# B&R Automation Studio project KeePakST401VersionX (part 2)

#### InverterFaultText.st - Implementation code
```iecst
(********************************************************************
 * COPYRIGHT --
 ********************************************************************
 * Program: ErrTxt
 * File: ErrTxt.st
 * Author: scoccimaroj
 * Created: November 09, 2010
 ********************************************************************
 * Implementation of function InverterFaultText
 ********************************************************************)

FUNCTION_BLOCK InverterFaultText

(*****************************************************************
		Initializing the Fault Tables
 ****************************************************************)

	IF ( isInitialized = FALSE) THEN
        (*ensure the fault table array creation is only run once upon start up*)
		isInitialized := TRUE;
        (*initialize internal fault comparison variable so that the first error is correctly written by the FUB *)
		PreviousFault :=  -1;
        (*initialize the output variable value*)
        LastFault := 0;
        (*this status will most likely not be seen by the FUB user but is written in case the table creation arrays are expanded enough for a visible delay to be seen*)
	    Status := INITIALIZING_ERROR_TEXT;

		(* Initialize the S44 Fault table first *)
		S44FaultTable[0].FaultNumber := 0;
		strcpy( ADR(S44FaultTable[0].FaultDescription), ADR('nOF - No Fault Present') );

		S44FaultTable[1].FaultNumber := 1;
		strcpy( ADR(S44FaultTable[1].FaultDescription), ADR('InF - Calibration Error') );

		S44FaultTable[2].FaultNumber := 3;
		strcpy( ADR(S44FaultTable[2].FaultDescription), ADR('CFF - Incorrect Configuration') );

		S44FaultTable[3].FaultNumber := 4;
		strcpy( ADR(S44FaultTable[3].FaultDescription), ADR('CFI - Invalid Configuration') );

		S44FaultTable[4].FaultNumber := 5;
		strcpy( ADR(S44FaultTable[4].FaultDescription), ADR('SLF1 - ModBus Communication Fault') );

		S44FaultTable[5].FaultNumber := 9;
		strcpy( ADR(S44FaultTable[5].FaultDescription), ADR('OCF - Over Current Fault') );

		S44FaultTable[6].FaultNumber := 10;
		strcpy( ADR(S44FaultTable[6].FaultDescription), ADR('CrF1 - Precharge Fault') );

		S44FaultTable[7].FaultNumber := 16;
		strcpy( ADR(S44FaultTable[7].FaultDescription), ADR('OHF - Drive Overheat') );

		S44FaultTable[8].FaultNumber := 17;
		strcpy( ADR(S44FaultTable[8].FaultDescription), ADR('OLF - Motor Overload') );

		S44FaultTable[9].FaultNumber := 18;
		strcpy( ADR(S44FaultTable[9].FaultDescription), ADR('ObF - Overbraking') );

		S44FaultTable[10].FaultNumber := 19;
		strcpy( ADR(S44FaultTable[10].FaultDescription), ADR('OSF - Mains Overvoltage') );

		S44FaultTable[11].FaultNumber := 20;
		strcpy( ADR(S44FaultTable[11].FaultDescription), ADR('OPF1 - 1 Output Phase Loss') );

		S44FaultTable[12].FaultNumber := 21;
		strcpy( ADR(S44FaultTable[12].FaultDescription), ADR('PHF - Input Phase Loss') );

		S44FaultTable[13].FaultNumber := 22;
		strcpy( ADR(S44FaultTable[13].FaultDescription), ADR('USF - Undervoltage') );

		S44FaultTable[14].FaultNumber := 23;
		strcpy( ADR(S44FaultTable[14].FaultDescription), ADR('SCF1 - Motor Short Circuit') );

		S44FaultTable[15].FaultNumber := 24;
		strcpy( ADR(S44FaultTable[15].FaultDescription), ADR('SOF - Overspeed') );

		S44FaultTable[16].FaultNumber := 25;
		strcpy( ADR(S44FaultTable[16].FaultDescription), ADR('tnF - Auto-tuning Fault') );

		S44FaultTable[17].FaultNumber := 26;
		strcpy( ADR(S44FaultTable[17].FaultDescription), ADR('InF1 - Rating Error') );

		S44FaultTable[18].FaultNumber := 27;
		strcpy( ADR(S44FaultTable[18].FaultDescription), ADR('InF2 - Power Calibration') );

		S44FaultTable[19].FaultNumber := 28;
		strcpy( ADR(S44FaultTable[19].FaultDescription), ADR('InF3 - Internal Serial Link') );

		S44FaultTable[20].FaultNumber := 29;
		strcpy( ADR(S44FaultTable[20].FaultDescription), ADR('InF4 - Internal Mfg area') );

		S44FaultTable[21].FaultNumber := 32;
		strcpy( ADR(S44FaultTable[21].FaultDescription), ADR('SCF3 - Ground Short Circuit') );

		S44FaultTable[22].FaultNumber := 33;
		strcpy( ADR(S44FaultTable[22].FaultDescription), ADR('OPF2 - 3 Output Phase Loss') );

		S44FaultTable[23].FaultNumber := 42;
		strcpy( ADR(S44FaultTable[23].FaultDescription), ADR('SLF2 - PowerSuite Communication') );

		S44FaultTable[24].FaultNumber := 45;
		strcpy( ADR(S44FaultTable[24].FaultDescription), ADR('SLF3 - HMI Communication Fault') );

		S44FaultTable[25].FaultNumber := 51;
		strcpy( ADR(S44FaultTable[25].FaultDescription), ADR('InF9 - Internal I measure') );

		S44FaultTable[26].FaultNumber := 53;
		strcpy( ADR(S44FaultTable[26].FaultDescription), ADR('InFb - Internal th. sensor') );

		S44FaultTable[27].FaultNumber := 54;
		strcpy( ADR(S44FaultTable[27].FaultDescription), ADR('tJF - IGBT Overheat') );

		S44FaultTable[28].FaultNumber := 55;
		strcpy( ADR(S44FaultTable[28].FaultDescription), ADR('SCF4 - IGBT Short Circuit') );

		S44FaultTable[29].FaultNumber := 56;
		strcpy( ADR(S44FaultTable[29].FaultDescription), ADR('SCF5 - Motor Short Circuit') );

		S44FaultTable[30].FaultNumber := 69;
		strcpy( ADR(S44FaultTable[30].FaultDescription), ADR('InFE - Internal CPU Fault') );

		S44FaultTable[31].FaultNumber := 77;
		strcpy( ADR(S44FaultTable[31].FaultDescription), ADR('CFI2') );

		S44FaultTable[32].FaultNumber := 100;
		strcpy( ADR(S44FaultTable[32].FaultDescription), ADR('ULF - Underload Fault') );

		S44FaultTable[33].FaultNumber := 101;
		strcpy( ADR(S44FaultTable[33].FaultDescription), ADR('OLC - Overload Fault') );

		S44FaultTable[34].FaultNumber := 106;
		strcpy( ADR(S44FaultTable[34].FaultDescription), ADR('LFF1') );

		S44FaultTable[35].FaultNumber := 253;
		strcpy( ADR(S44FaultTable[35].FaultDescription), ADR('XXXX') );

		(* Initialize the X64 Table *)
		X64FaultTable[0].FaultNumber := 0;
		strcpy( ADR(X64FaultTable[0].FaultDescription), ADR('nOF - No Fault Code') );

		X64FaultTable[1].FaultNumber := 3;
		strcpy( ADR(X64FaultTable[1].FaultDescription), ADR('CFF - Incorrect Configuration') );

		X64FaultTable[2].FaultNumber := 4;
		strcpy( ADR(X64FaultTable[2].FaultDescription), ADR('CFI - Invalid Configuration') );

		X64FaultTable[3].FaultNumber := 5;
		strcpy( ADR(X64FaultTable[3].FaultDescription), ADR('SLF - Communication Fault') );

		X64FaultTable[4].FaultNumber := 6;
		strcpy( ADR(X64FaultTable[4].FaultDescription), ADR('ILF - Internal Communication Interuption') );

		X64FaultTable[5].FaultNumber := 7;
		strcpy( ADR(X64FaultTable[5].FaultDescription), ADR('CnF - Communication Option Card') );

		X64FaultTable[6].FaultNumber := 8;
		strcpy( ADR(X64FaultTable[6].FaultDescription), ADR('EPF - External Fault') );

		X64FaultTable[7].FaultNumber := 9;
		strcpy( ADR(X64FaultTable[7].FaultDescription), ADR('OCF - Overcurrent') );

		X64FaultTable[8].FaultNumber := 10;
		strcpy( ADR(X64FaultTable[8].FaultDescription), ADR('CrF - Capacitor pre-charge') );

		X64FaultTable[9].FaultNumber := 13;
		strcpy( ADR(X64FaultTable[9].FaultDescription), ADR('LFF - 4 - 20 mA loss') );

		X64FaultTable[10].FaultNumber := 16;
		strcpy( ADR(X64FaultTable[10].FaultDescription), ADR('OHF - Drive Overheating') );

		X64FaultTable[11].FaultNumber := 17;
		strcpy( ADR(X64FaultTable[11].FaultDescription), ADR('OLF - Motor Overload') );

		X64FaultTable[12].FaultNumber := 18;
		strcpy( ADR(X64FaultTable[12].FaultDescription), ADR('ObF - DC Bus Overvoltage') );

		X64FaultTable[13].FaultNumber := 19;
		strcpy( ADR(X64FaultTable[13].FaultDescription), ADR('OSF - Line Supply Overvoltage') );

		X64FaultTable[14].FaultNumber := 20;
		strcpy( ADR(X64FaultTable[14].FaultDescription), ADR('OPF - Motor Phase Lose') );

		X64FaultTable[15].FaultNumber := 21;
		strcpy( ADR(X64FaultTable[15].FaultDescription), ADR('PHF - Line Phase Loss') );

		X64FaultTable[16].FaultNumber := 22;
		strcpy( ADR(X64FaultTable[16].FaultDescription), ADR('USF - Line Supply Undervoltage') );

		X64FaultTable[17].FaultNumber := 23;
		strcpy( ADR(X64FaultTable[17].FaultDescription), ADR('OCF - Motor Short Circuit (phase to phase)') );

		X64FaultTable[18].FaultNumber := 24;
		strcpy( ADR(X64FaultTable[18].FaultDescription), ADR('SOF - Motor Overspeed') );

		X64FaultTable[19].FaultNumber := 25;
		strcpy( ADR(X64FaultTable[19].FaultDescription), ADR('tnF - Auto-tuning was unsuccessful') );

		X64FaultTable[20].FaultNumber := 26;
		strcpy( ADR(X64FaultTable[20].FaultDescription), ADR('IF1 - Unknow rating') );

		X64FaultTable[21].FaultNumber := 27;
		strcpy( ADR(X64FaultTable[21].FaultDescription), ADR('IF2 - MMI card') );

		X64FaultTable[22].FaultNumber := 28;
		strcpy( ADR(X64FaultTable[22].FaultDescription), ADR('IF3 - MMI communication') );

		X64FaultTable[23].FaultNumber := 29;
		strcpy( ADR(X64FaultTable[23].FaultDescription), ADR('IF4 - Industrial EEPROM memory') );

		X64FaultTable[24].FaultNumber := 30;
		strcpy( ADR(X64FaultTable[24].FaultDescription), ADR('EEF - EEPROM memory') );

		X64FaultTable[25].FaultNumber := 31;
		strcpy( ADR(X64FaultTable[25].FaultDescription), ADR('OCF - Impeding Short Circuit') );

		X64FaultTable[26].FaultNumber := 32;
		strcpy( ADR(X64FaultTable[26].FaultDescription), ADR('SCF - Motor Short Circuit (to ground)') );

		X64FaultTable[27].FaultNumber := 33;
		strcpy( ADR(X64FaultTable[27].FaultDescription), ADR('OPF - Motor Phase Loss - 3 phases') );

		X64FaultTable[28].FaultNumber := 34;
		strcpy( ADR(X64FaultTable[28].FaultDescription), ADR('COF - Communication Interuption') );

		X64FaultTable[29].FaultNumber := 35;
		strcpy( ADR(X64FaultTable[29].FaultDescription), ADR('bLF - Brake Control') );

		X64FaultTable[30].FaultNumber := 36;
		strcpy( ADR(X64FaultTable[30].FaultDescription), ADR('OCF - Power Module on 15 kW drive') );

		X64FaultTable[31].FaultNumber := 55;
		strcpy( ADR(X64FaultTable[31].FaultDescription), ADR('SCF - Power Module or Motor Short Circuit') );

		(* Initialize the P84 Table *)
		P84FaultTable[0].FaultNumber := 0;
		strcpy( ADR(P84FaultTable[0].FaultDescription), ADR('nOF - No Fault') );

		P84FaultTable[1].FaultNumber := 1;
		strcpy( ADR(P84FaultTable[1].FaultDescription), ADR('InF - Calibration Error') );

		P84FaultTable[2].FaultNumber := 2;
		strcpy( ADR(P84FaultTable[2].FaultDescription), ADR('EEF1 - Control EEPROM') );

		P84FaultTable[3].FaultNumber := 3;
		strcpy( ADR(P84FaultTable[3].FaultDescription), ADR('CFF - Incorrect Configuration') );

		P84FaultTable[4].FaultNumber := 4;
		strcpy( ADR(P84FaultTable[4].FaultDescription), ADR('CFI - Invalid Configuration') );

		P84FaultTable[5].FaultNumber := 5;
		strcpy( ADR(P84FaultTable[5].FaultDescription), ADR('SLF1 - Communication Error') );

		P84FaultTable[6].FaultNumber := 6;
		strcpy( ADR(P84FaultTable[6].FaultDescription), ADR('ILF - Internal Communication Link') );

		P84FaultTable[7].FaultNumber := 7;
		strcpy( ADR(P84FaultTable[7].FaultDescription), ADR('CnF - Communication Network') );

		P84FaultTable[8].FaultNumber := 8;
		strcpy( ADR(P84FaultTable[8].FaultDescription), ADR('EPF1 - External Fault') );

		P84FaultTable[9].FaultNumber := 9;
		strcpy( ADR(P84FaultTable[9].FaultDescription), ADR('OCF - Overcurrent') );

		P84FaultTable[10].FaultNumber := 10;
		strcpy( ADR(P84FaultTable[10].FaultDescription), ADR('CrF - Precharge') );

		P84FaultTable[11].FaultNumber := 11;
		strcpy( ADR(P84FaultTable[11].FaultDescription), ADR('SPF - Speed Feedback loss') );

		P84FaultTable[12].FaultNumber := 12;
		strcpy( ADR(P84FaultTable[12].FaultDescription), ADR('AnF - Load Slipping') );

		P84FaultTable[13].FaultNumber := 13;
		strcpy( ADR(P84FaultTable[13].FaultDescription), ADR('LFF2 - AI2 4-20 mA Loss') );

		P84FaultTable[14].FaultNumber := 14;
		strcpy( ADR(P84FaultTable[14].FaultDescription), ADR('PtF1 - PTC1 Probe') );

		P84FaultTable[15].FaultNumber := 15;
		strcpy( ADR(P84FaultTable[15].FaultDescription), ADR('OtF1 - PTC1 Overheat') );

		P84FaultTable[16].FaultNumber := 16;
		strcpy( ADR(P84FaultTable[16].FaultDescription), ADR('OHF - Drive Overheat') );

		P84FaultTable[17].FaultNumber := 17;
		strcpy( ADR(P84FaultTable[17].FaultDescription), ADR('OLF - Motor Overload') );

		P84FaultTable[18].FaultNumber := 18;
		strcpy( ADR(P84FaultTable[18].FaultDescription), ADR('ObF - Overbraking') );

		P84FaultTable[19].FaultNumber := 19;
		strcpy( ADR(P84FaultTable[19].FaultDescription), ADR('OSF - Mains Overvoltage') );

		P84FaultTable[20].FaultNumber := 20;
		strcpy( ADR(P84FaultTable[20].FaultDescription), ADR('OPF1 - 1 Output Phase Loss') );

		P84FaultTable[21].FaultNumber := 21;
		strcpy( ADR(P84FaultTable[21].FaultDescription), ADR('PHF - Input Phase Loss') );

		P84FaultTable[22].FaultNumber := 22;
		strcpy( ADR(P84FaultTable[22].FaultDescription), ADR('USF - Undervoltage') );

		P84FaultTable[23].FaultNumber := 23;
		strcpy( ADR(P84FaultTable[23].FaultDescription), ADR('SCF1 - Motor Short Circuit') );

		P84FaultTable[24].FaultNumber := 24;
		strcpy( ADR(P84FaultTable[24].FaultDescription), ADR('SOF - Overspeed') );

		P84FaultTable[25].FaultNumber := 25;
		strcpy( ADR(P84FaultTable[25].FaultDescription), ADR('tnF - Auto-tuning Unsuccessful') );

		P84FaultTable[26].FaultNumber := 26;
		strcpy( ADR(P84FaultTable[26].FaultDescription), ADR('InF1 - Rating Error') );

		P84FaultTable[27].FaultNumber := 27;
		strcpy( ADR(P84FaultTable[27].FaultDescription), ADR('InF2 - Power Calibration') );

		P84FaultTable[28].FaultNumber := 28;
		strcpy( ADR(P84FaultTable[28].FaultDescription), ADR('InF3 - Internal Serial Link') );

		P84FaultTable[29].FaultNumber := 29;
		strcpy( ADR(P84FaultTable[29].FaultDescription), ADR('InF4 - Internal Mfg Area') );

		P84FaultTable[30].FaultNumber := 30;
		strcpy( ADR(P84FaultTable[30].FaultDescription), ADR('EEF2 - Power EEPROM') );

		P84FaultTable[31].FaultNumber := 31;
		strcpy( ADR(P84FaultTable[31].FaultDescription), ADR('SCF2 - Impedant Short Circuit') );

		P84FaultTable[32].FaultNumber := 32;
		strcpy( ADR(P84FaultTable[32].FaultDescription), ADR('SCF3 - Ground Short Circuit') );

		P84FaultTable[33].FaultNumber := 33;
		strcpy( ADR(P84FaultTable[33].FaultDescription), ADR('OPF2 - 3 Phase Output Loss') );

		P84FaultTable[34].FaultNumber := 34;
		strcpy( ADR(P84FaultTable[34].FaultDescription), ADR('COF - Powerlink Communication') );

		P84FaultTable[35].FaultNumber := 35;
		strcpy( ADR(P84FaultTable[35].FaultDescription), ADR('bLF - Brake Control') );

		P84FaultTable[36].FaultNumber := 37;
		strcpy( ADR(P84FaultTable[36].FaultDescription), ADR('InF7 - Internal Hard Init') );

		P84FaultTable[37].FaultNumber := 38;
		strcpy( ADR(P84FaultTable[37].FaultDescription), ADR('EPF2 - External Fault Com.') );

		P84FaultTable[38].FaultNumber := 39;
		strcpy( ADR(P84FaultTable[38].FaultDescription), ADR('APF - Application Fault') );

		P84FaultTable[39].FaultNumber := 40;
		strcpy( ADR(P84FaultTable[39].FaultDescription), ADR('InF8 - Internal Ctrl Supply') );

		P84FaultTable[40].FaultNumber := 41;
		strcpy( ADR(P84FaultTable[40].FaultDescription), ADR('brF - Brake Feedback') );

		P84FaultTable[41].FaultNumber := 42;
		strcpy( ADR(P84FaultTable[41].FaultDescription), ADR('SLF2 - PowerSuite Communication.') );

		P84FaultTable[42].FaultNumber := 43;
		strcpy( ADR(P84FaultTable[42].FaultDescription), ADR('ECF - Encoder Coupling') );

		P84FaultTable[43].FaultNumber := 44;
		strcpy( ADR(P84FaultTable[43].FaultDescription), ADR('SSF - Torque Current Limit') );

		P84FaultTable[44].FaultNumber :=45 ;
		strcpy( ADR(P84FaultTable[44].FaultDescription), ADR('SLF3 - HMI com.') );

		P84FaultTable[45].FaultNumber := 46;
		strcpy( ADR(P84FaultTable[45].FaultDescription), ADR('PrF - Power Removal') );

		P84FaultTable[46].FaultNumber := 47;
		strcpy( ADR(P84FaultTable[46].FaultDescription), ADR('PtF2 - PTC2 Probe') );

		P84FaultTable[47].FaultNumber := 48;
		strcpy( ADR(P84FaultTable[47].FaultDescription), ADR('OtF2 - PTC2 Overheat') );

		P84FaultTable[48].FaultNumber := 49;
		strcpy( ADR(P84FaultTable[48].FaultDescription), ADR('PtFL - LI6=PTC Probe') );

		P84FaultTable[49].FaultNumber := 50;
		strcpy( ADR(P84FaultTable[49].FaultDescription), ADR('OtFL - PTC Fault') );

		P84FaultTable[50].FaultNumber := 51;
		strcpy( ADR(P84FaultTable[50].FaultDescription), ADR('InF9 - Internal I measure') );

		P84FaultTable[51].FaultNumber := 52;
		strcpy( ADR(P84FaultTable[51].FaultDescription), ADR('InFA - Internal Mains Circuit') );

		P84FaultTable[52].FaultNumber := 53;
		strcpy( ADR(P84FaultTable[52].FaultDescription), ADR('InFb - Internal th. Sensor') );

		P84FaultTable[53].FaultNumber := 54;
		strcpy( ADR(P84FaultTable[53].FaultDescription), ADR('tJF - IGBT Overheat') );

		P84FaultTable[54].FaultNumber := 55;
		strcpy( ADR(P84FaultTable[54].FaultDescription), ADR('SCF4 - IGBT Short Circuit') );

		P84FaultTable[55].FaultNumber := 56;
		strcpy( ADR(P84FaultTable[55].FaultDescription), ADR('SCF5 - Motor Short Circuit') );

		P84FaultTable[56].FaultNumber :=57 ;
		strcpy( ADR(P84FaultTable[56].FaultDescription), ADR('SrF - Torque Time-out') );

		P84FaultTable[57].FaultNumber := 58;
		strcpy( ADR(P84FaultTable[57].FaultDescription), ADR('FCF1 - Output Contact Stuck') );

		P84FaultTable[58].FaultNumber := 59;
		strcpy( ADR(P84FaultTable[58].FaultDescription), ADR('FCF2 - Output Contact Open') );

		P84FaultTable[59].FaultNumber := 60;
		strcpy( ADR(P84FaultTable[59].FaultDescription), ADR('InFC - Int. T Measurement') );

		P84FaultTable[60].FaultNumber := 61;
		strcpy( ADR(P84FaultTable[60].FaultDescription), ADR('AI2F - AI2 Input') );

		P84FaultTable[61].FaultNumber := 62;
		strcpy( ADR(P84FaultTable[61].FaultDescription), ADR('EnF - Encoder') );

		P84FaultTable[62].FaultNumber := 63;
		strcpy( ADR(P84FaultTable[62].FaultDescription), ADR('CrF2 - Thyr. Soft Charge') );

		P84FaultTable[63].FaultNumber := 64;
		strcpy( ADR(P84FaultTable[63].FaultDescription), ADR('LCF - Input Contactor') );

		P84FaultTable[64].FaultNumber := 65;
		strcpy( ADR(P84FaultTable[64].FaultDescription), ADR('bUF - DB Unit Short Circuit') );

		P84FaultTable[65].FaultNumber := 66;
		strcpy( ADR(P84FaultTable[65].FaultDescription), ADR('dCF - Iff. I Fault') );

		P84FaultTable[66].FaultNumber := 67;
		strcpy( ADR(P84FaultTable[66].FaultDescription), ADR('HdF - IGBT  Desaturation') );

		P84FaultTable[67].FaultNumber := 68;
		strcpy( ADR(P84FaultTable[67].FaultDescription), ADR('InF6 - Internal Option') );

		P84FaultTable[68].FaultNumber := 69;
		strcpy( ADR(P84FaultTable[68].FaultDescription), ADR('InFE - Internal CPU') );

		P84FaultTable[69].FaultNumber := 70;
		strcpy( ADR(P84FaultTable[69].FaultDescription), ADR('bOF - BR Overload') );

		P84FaultTable[70].FaultNumber := 71;
		strcpy( ADR(P84FaultTable[70].FaultDescription), ADR('LFF3 - AI3 4-20 mA Loss') );

		P84FaultTable[71].FaultNumber := 72;
		strcpy( ADR(P84FaultTable[71].FaultDescription), ADR('LEF4 - AI4 4-20 mA Loss') );

		P84FaultTable[72].FaultNumber := 73;
		strcpy( ADR(P84FaultTable[72].FaultDescription), ADR('HCF - Cards Pairing') );

		P84FaultTable[73].FaultNumber := 76;
		strcpy( ADR(P84FaultTable[73].FaultDescription), ADR('dLF - Load Fault') );

		P84FaultTable[74].FaultNumber := 99;
		strcpy( ADR(P84FaultTable[74].FaultDescription), ADR('CSF - Ch. SW. Fault') );

		(* Initialize the P74 Table *)
		P74FaultTable[0].FaultNumber := 0;
		strcpy( ADR(P74FaultTable[0].FaultDescription), ADR('nOF - No Fault') );

		P74FaultTable[1].FaultNumber := 1;
		strcpy( ADR(P74FaultTable[1].FaultDescription), ADR('InF - Calibration Error') );

		P74FaultTable[2].FaultNumber := 2;
		strcpy( ADR(P74FaultTable[2].FaultDescription), ADR('EEF1 - Control EEPROM') );

		P74FaultTable[3].FaultNumber := 3;
		strcpy( ADR(P74FaultTable[3].FaultDescription), ADR('CFF - Incorrect Configuration') );

		P74FaultTable[4].FaultNumber := 4;
		strcpy( ADR(P74FaultTable[4].FaultDescription), ADR('CFI - Invalid Configuration') );

		P74FaultTable[5].FaultNumber := 5;
		strcpy( ADR(P74FaultTable[5].FaultDescription), ADR('SLF1 - Communication Error') );

		P74FaultTable[6].FaultNumber := 6;
		strcpy( ADR(P74FaultTable[6].FaultDescription), ADR('ILF - Internal Communication Link') );

		P74FaultTable[7].FaultNumber := 7;
		strcpy( ADR(P74FaultTable[7].FaultDescription), ADR('CnF - Communication Network') );

		P74FaultTable[8].FaultNumber := 8;
		strcpy( ADR(P74FaultTable[8].FaultDescription), ADR('EPF1 - External Fault') );

		P74FaultTable[9].FaultNumber := 9;
		strcpy( ADR(P74FaultTable[9].FaultDescription), ADR('OCF - Overcurrent') );

		P74FaultTable[10].FaultNumber := 10;
		strcpy( ADR(P74FaultTable[10].FaultDescription), ADR('CrF - Precharge') );

		P74FaultTable[11].FaultNumber := 11;
		strcpy( ADR(P74FaultTable[11].FaultDescription), ADR('SPF - Speed Feedback loss') );

		P74FaultTable[12].FaultNumber := 16;
		strcpy( ADR(P74FaultTable[12].FaultDescription), ADR('OHF - Drive Overheat') );

		P74FaultTable[13].FaultNumber := 17;
		strcpy( ADR(P74FaultTable[13].FaultDescription), ADR('OLF - Motor Overload') );

		P74FaultTable[14].FaultNumber := 18;
		strcpy( ADR(P74FaultTable[14].FaultDescription), ADR('ObF - Overbraking') );

		P74FaultTable[15].FaultNumber := 19;
		strcpy( ADR(P74FaultTable[15].FaultDescription), ADR('OSF - Mains Overvoltage') );

		P74FaultTable[16].FaultNumber := 20;
		strcpy( ADR(P74FaultTable[16].FaultDescription), ADR('OPF1 - 1 Output Phase Loss') );

		P74FaultTable[17].FaultNumber := 21;
		strcpy( ADR(P74FaultTable[17].FaultDescription), ADR('PHF - Input Phase Loss') );

		P74FaultTable[18].FaultNumber := 22;
		strcpy( ADR(P74FaultTable[18].FaultDescription), ADR('USF - Undervoltage') );

		P74FaultTable[19].FaultNumber := 23;
		strcpy( ADR(P74FaultTable[19].FaultDescription), ADR('SCF1 - Motor Short Circuit') );

		P74FaultTable[20].FaultNumber := 24;
		strcpy( ADR(P74FaultTable[20].FaultDescription), ADR('SOF - Overspeed') );

		P74FaultTable[21].FaultNumber := 25;
		strcpy( ADR(P74FaultTable[21].FaultDescription), ADR('tnF - Auto-tuning Unsuccessful') );

		P74FaultTable[22].FaultNumber := 26;
		strcpy( ADR(P74FaultTable[22].FaultDescription), ADR('InF1 - Rating Error') );

		P74FaultTable[23].FaultNumber := 27;
		strcpy( ADR(P74FaultTable[23].FaultDescription), ADR('InF2 - Power Calibration') );

		P74FaultTable[24].FaultNumber := 28;
		strcpy( ADR(P74FaultTable[24].FaultDescription), ADR('InF3 - Internal Serial Link') );

		P74FaultTable[25].FaultNumber := 29;
		strcpy( ADR(P74FaultTable[25].FaultDescription), ADR('InF4 - Internal Mfg Area') );

		P74FaultTable[26].FaultNumber := 30;
		strcpy( ADR(P74FaultTable[26].FaultDescription), ADR('EEF2 - Power EEPROM') );

		P74FaultTable[27].FaultNumber := 31;
		strcpy( ADR(P74FaultTable[27].FaultDescription), ADR('SCF2 - Impedant Short Circuit') );

		P74FaultTable[28].FaultNumber := 32;
		strcpy( ADR(P74FaultTable[28].FaultDescription), ADR('SCF3 - Ground Short Circuit') );

		P74FaultTable[29].FaultNumber := 33;
		strcpy( ADR(P74FaultTable[29].FaultDescription), ADR('OPF2 - 3 Phase Output Loss') );

		P74FaultTable[30].FaultNumber := 34;
		strcpy( ADR(P74FaultTable[30].FaultDescription), ADR('COF - Powerlink Communication') );

		P74FaultTable[31].FaultNumber := 35;
		strcpy( ADR(P74FaultTable[31].FaultDescription), ADR('bLF - Brake Control') );

		P74FaultTable[32].FaultNumber := 38;
		strcpy( ADR(P74FaultTable[32].FaultDescription), ADR('EPF2 - External Fault Com.') );

		P74FaultTable[33].FaultNumber := 41;
		strcpy( ADR(P74FaultTable[33].FaultDescription), ADR('brF - Brake Feedback') );

		P74FaultTable[34].FaultNumber := 42;
		strcpy( ADR(P74FaultTable[34].FaultDescription), ADR('SLF2 - PowerSuite Communication.') );

		P74FaultTable[35].FaultNumber := 43;
		strcpy( ADR(P74FaultTable[35].FaultDescription), ADR('ECF - Encoder Coupling') );

		P74FaultTable[36].FaultNumber := 44;
		strcpy( ADR(P74FaultTable[36].FaultDescription), ADR('SSF - Torque Current Limit') );

		P74FaultTable[37].FaultNumber := 45 ;
		strcpy( ADR(P74FaultTable[37].FaultDescription), ADR('SLF3 - HMI com.') );

		P74FaultTable[38].FaultNumber := 46;
		strcpy( ADR(P74FaultTable[38].FaultDescription), ADR('PrF - Power Removal') );

		P74FaultTable[39].FaultNumber := 49;
		strcpy( ADR(P74FaultTable[39].FaultDescription), ADR('PtFL - LI6=PTC Probe') );

		P74FaultTable[40].FaultNumber := 50;
		strcpy( ADR(P74FaultTable[40].FaultDescription), ADR('OtFL - PTC Fault') );

		P74FaultTable[41].FaultNumber := 51;
		strcpy( ADR(P74FaultTable[41].FaultDescription), ADR('InF9 - Internal I measure') );

		P74FaultTable[42].FaultNumber := 52;
		strcpy( ADR(P74FaultTable[42].FaultDescription), ADR('InFA - Internal Mains Circuit') );

		P74FaultTable[43].FaultNumber := 53;
		strcpy( ADR(P74FaultTable[43].FaultDescription), ADR('InFb - Internal th. Sensor') );

		P74FaultTable[44].FaultNumber := 54;
		strcpy( ADR(P74FaultTable[44].FaultDescription), ADR('tJF - IGBT Overheat') );

		P74FaultTable[45].FaultNumber := 55;
		strcpy( ADR(P74FaultTable[45].FaultDescription), ADR('SCF4 - IGBT Short Circuit') );

		P74FaultTable[46].FaultNumber := 56;
		strcpy( ADR(P74FaultTable[46].FaultDescription), ADR('SCF5 - Motor Short Circuit') );

		P74FaultTable[47].FaultNumber := 57 ;
		strcpy( ADR(P74FaultTable[47].FaultDescription), ADR('SrF - Torque Time-out') );

		P74FaultTable[48].FaultNumber := 58;
		strcpy( ADR(P74FaultTable[48].FaultDescription), ADR('FCF1 - Output Contact Stuck') );

		P74FaultTable[49].FaultNumber := 59;
		strcpy( ADR(P74FaultTable[49].FaultDescription), ADR('FCF2 - Output Contact Open') );

		P74FaultTable[50].FaultNumber := 61;
		strcpy( ADR(P74FaultTable[50].FaultDescription), ADR('AI2F - AI2 Input') );

		P74FaultTable[51].FaultNumber := 64;
		strcpy( ADR(P74FaultTable[51].FaultDescription), ADR('LCF - Input Contactor') );

		P74FaultTable[52].FaultNumber := 66;
		strcpy( ADR(P74FaultTable[52].FaultDescription), ADR('dCF - Iff. I Fault') );

		P74FaultTable[53].FaultNumber := 67;
		strcpy( ADR(P74FaultTable[53].FaultDescription), ADR('HdF - IGBT  Desaturation') );

		P74FaultTable[54].FaultNumber := 68;
		strcpy( ADR(P74FaultTable[54].FaultDescription), ADR('InF6 - Internal Option') );

		P74FaultTable[55].FaultNumber := 69;
		strcpy( ADR(P74FaultTable[55].FaultDescription), ADR('InFE - Internal CPU') );

		P74FaultTable[56].FaultNumber := 71;
		strcpy( ADR(P74FaultTable[56].FaultDescription), ADR('LFF3 - AI3 4-20 mA Loss') );

		P74FaultTable[57].FaultNumber := 73;
		strcpy( ADR(P74FaultTable[57].FaultDescription), ADR('HCF - Cards Pairing') );

		P74FaultTable[58].FaultNumber := 76;
		strcpy( ADR(P74FaultTable[58].FaultDescription), ADR('dLF - Load Fault') );

		P74FaultTable[59].FaultNumber := 77;
		strcpy( ADR(P74FaultTable[59].FaultDescription), ADR('CFI2 - Bad Configuration') );

		P74FaultTable[60].FaultNumber := 99;
		strcpy( ADR(P74FaultTable[60].FaultDescription), ADR('CSF - Ch. SW. Fault') );

		P74FaultTable[61].FaultNumber := 100;
		strcpy( ADR(P74FaultTable[61].FaultDescription), ADR('ULF - Pr. Underload Fault') );

		P74FaultTable[62].FaultNumber := 101;
		strcpy( ADR(P74FaultTable[62].FaultDescription), ADR('OLC - Proc. Overload Fault') );

		P74FaultTable[63].FaultNumber := 105;
		strcpy( ADR(P74FaultTable[63].FaultDescription), ADR('ASF - Angle Error') );

		P74FaultTable[64].FaultNumber := 107;
		strcpy( ADR(P74FaultTable[64].FaultDescription), ADR('SAFF - Safety Fault') );

		P74FaultTable[65].FaultNumber := 108;
		strcpy( ADR(P74FaultTable[65].FaultDescription), ADR('FbE - FB Fault') );

		P74FaultTable[66].FaultNumber := 109;
		strcpy( ADR(P74FaultTable[66].FaultDescription), ADR('FbES - FB Stop Fault') );
	ELSE
        (*this status will only be seen if the initialization of the fualt text arrays fails*)
        Status := INACTIVE;
	END_IF

	(* End of initializing the tables *)

	(*****************************************************
	Getting the Fault Text
	*****************************************************)
    IF isInitialized = TRUE THEN
        (* Do the search for a S44 drive *)
        IF (DriveType = EACPInverter_S44) THEN

            (*Cyclically write the internal previous fault number into the output variable LastFault*)
            LastFault := PreviousFault;

            IF Execute = TRUE THEN
                Status := BUSY;
                (* Only do a look up if a new fault number occured *)
                IF ( PreviousFault <> FaultNumber ) THEN
                    PreviousFault := FaultNumber;

                    (* Clear out the text in the fault string *)
                    strcpy(FaultText, ADR('') );

                    FOR i:= 0 TO 35 BY 1 DO
                        IF (FaultNumber = S44FaultTable[i].FaultNumber) THEN
                            strcpy(FaultText, ADR(S44FaultTable[i].FaultDescription) );
                            EXIT;
                        END_IF;
                    END_FOR;
                END_IF;
            ELSE
                Status := IDLE;
            END_IF;
            (* Do the search for a X64 drive *)
        ELSIF (DriveType = EACPInverter_X64) THEN

            (*Cyclically write the internal previous fault number into the output variable LastFault*)
            LastFault := PreviousFault;

            IF Execute = TRUE THEN
                Status := BUSY;
                (* Only do a look up if a new fault number occured *)
                IF ( PreviousFault <> FaultNumber ) THEN
                    PreviousFault := FaultNumber;

                    (* Clear out the text in the fault string *)
                    strcpy(FaultText, ADR('') );

                    FOR i:= 0 TO 31 BY 1 DO
                        IF (FaultNumber = X64FaultTable[i].FaultNumber) THEN
                            strcpy(FaultText, ADR(X64FaultTable[i].FaultDescription) );
                            EXIT;
                        END_IF;
                    END_FOR;
                END_IF;
            ELSE
                Status := IDLE;
            END_IF;

            (* Do the search for a P84 drive *)
        ELSIF (DriveType = EACPInverter_P84) THEN

            (*Cyclically write the internal previous fault number into the output variable LastFault*)
            LastFault := PreviousFault;

            IF Execute = TRUE THEN
                Status := BUSY;
                (* Only do a look up if a new fault number occured *)
                IF ( PreviousFault <> FaultNumber ) THEN
                    PreviousFault := FaultNumber;

                    (* Clear out the text in the fault string *)
                    strcpy(FaultText, ADR('') );

                    FOR i:= 0 TO 74 BY 1 DO
                        IF (FaultNumber = P84FaultTable[i].FaultNumber) THEN
                            strcpy(FaultText, ADR(P84FaultTable[i].FaultDescription) );
                            EXIT;
                        END_IF;
                    END_FOR;
                END_IF;
            ELSE
                Status := IDLE;
            END_IF;

        ELSIF (DriveType = EACPInverter_P74) THEN

            (*Cyclically write the internal previous fault number into the output variable LastFault*)
            LastFault := PreviousFault;

            IF Execute = TRUE THEN
                Status := BUSY;
                (* Only do a look up if a new fault number occured *)
                IF ( PreviousFault <> FaultNumber ) THEN
                    PreviousFault := FaultNumber;

                    (* Clear out the text in the fault string *)
                    strcpy(FaultText, ADR('') );

                    FOR i:= 0 TO 66 BY 1 DO
                        IF (FaultNumber = P74FaultTable[i].FaultNumber) THEN
                            strcpy(FaultText, ADR(P74FaultTable[i].FaultDescription) );
                            EXIT;
                        END_IF	;
                    END_FOR	;
                END_IF;
            ELSE
                Status := IDLE;
            END_IF;

        END_IF;
    END_IF;

END_FUNCTION_BLOCK
```

### Library Logical/Libraries/DistCalc (ANSIC)

#### DistCalc.fun - Exported functions and function blocks
```iecst
FUNCTION DetermineDistanceToStopPos : REAL (*TODO: Add your comment here*) (*$GROUP=User,$CAT=User,$GROUPICON=User.png,$CATICON=User.png*)
	VAR_INPUT
		EncoderPos : REAL;
		StopPos : REAL;
	END_VAR
END_FUNCTION
```

#### DetermineDistanceToStopPos.c
```c
#include <bur/plctypes.h>
#include <math.h>
#ifdef __cplusplus
	extern "C"
	{
#endif
	#include "DistCalc.h"
#ifdef __cplusplus
	};
#endif
/* TODO: Add your comment here */
REAL DetermineDistanceToStopPos(float EncoderPos, float StopPos)
{
	REAL diff = 0.0;
	REAL modDiff = 0.0;

	diff = fabs(EncoderPos - StopPos);

	modDiff = fmod(diff,360.0);

	return (180.0 - fabs(modDiff - 180.0));

}
```

### Library Logical/Libraries/MappCall (IEC)
Depends on: Types

#### Constants.var - Exported constants
```iecst
VAR CONSTANT
	HOME_SEARCH_SPEED : REAL := 20;
	SENSOR_OFFSET : REAL := 2;
END_VAR
```

#### MappCall.fun - Exported functions and function blocks
```iecst
{REDUND_ERROR} FUNCTION_BLOCK AxisBasic (*Implements config and basic for a mapp axis*) (*$GROUP=User,$CAT=User,$GROUPICON=User.png,$CATICON=User.png*)
	VAR_INPUT
		pMpLink : UDINT;
		pAxis : UDINT;
		pEndlessPosition : {REDUND_UNREPLICABLE} UDINT;
		AxisInterface : REFERENCE TO Axis_Interface_typ;
		OdometerValue : LREAL;
		Override : REAL;
		ErrorReset : BOOL;
	END_VAR
	VAR
		AxisBasic : {REDUND_UNREPLICABLE} MpAxisBasic;
		AxisConfig : MpAxisBasicConfig;
		AbsDistance : LREAL;
		zzInternalMemory : ARRAY[0..40] OF SINT; (*Internal memory*)
		SetOverride : MC_SetOverride;
	END_VAR
END_FUNCTION_BLOCK
```

#### AxisBasic.ld
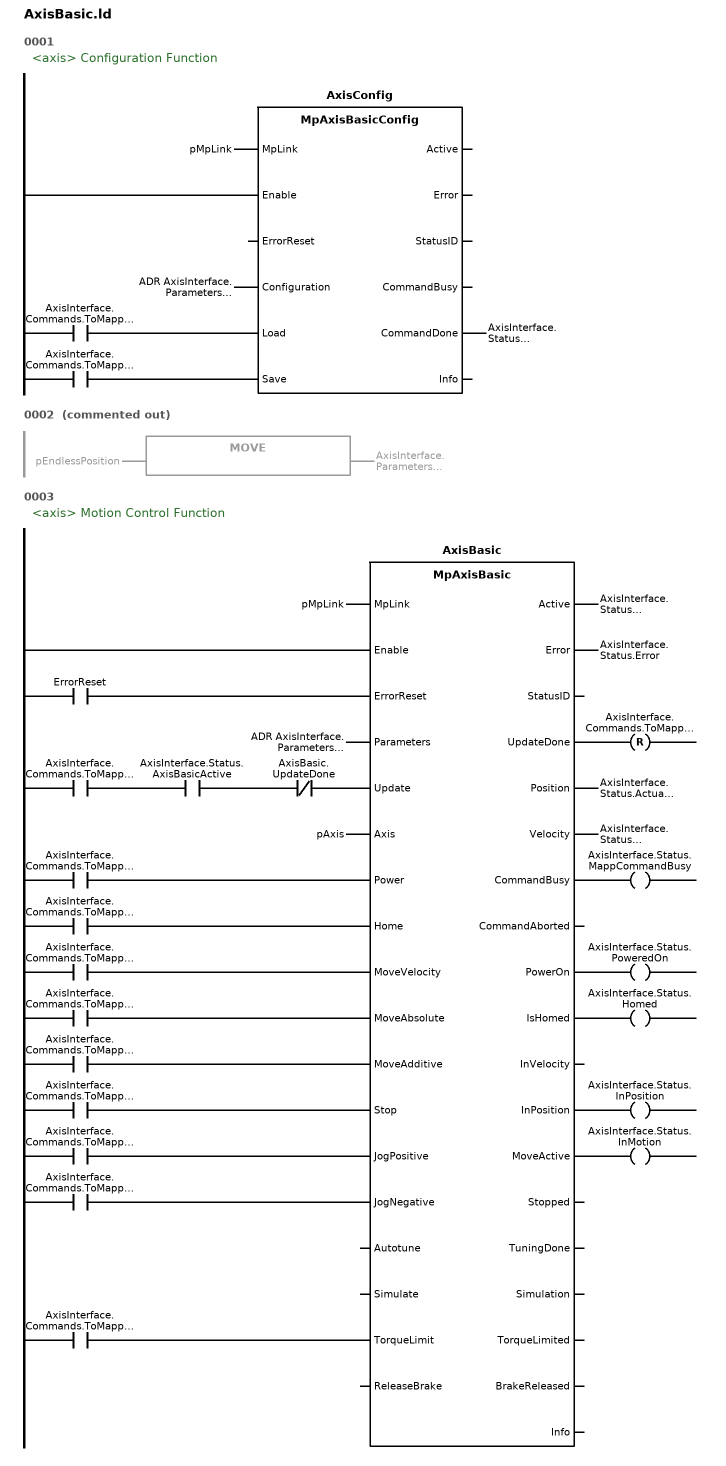
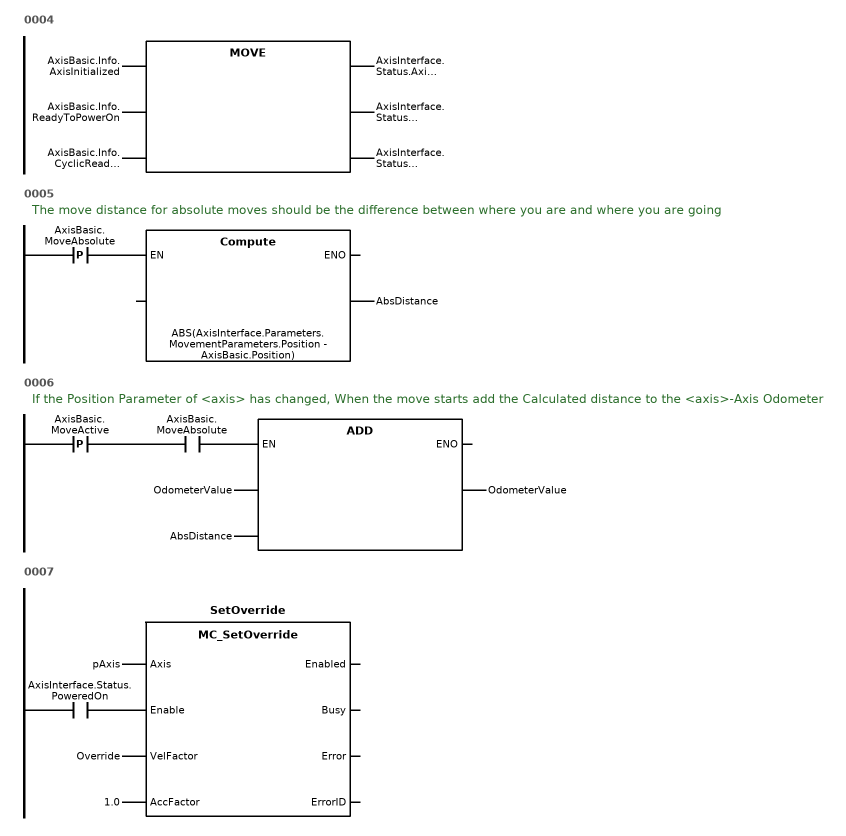
Ladder, written as Structured Text:
```iecst
(* Implements config and basic for a mapp axis *)
FUNCTION_BLOCK AxisBasic
VAR
    _e1 : R_TRIG;
    _e2 : R_TRIG;
END_VAR
(* Network 1: <axis> Configuration Function *)
AxisConfig(MpLink := pMpLink, Enable := TRUE, Configuration := ADR(AxisInterface.Parameters.AxisAndDrivePars), Load := AxisInterface.Commands.ToMapp.LoadConfig, Save := AxisInterface.Commands.ToMapp.SaveConfig);
AxisInterface.Status.ConfigCommandDone := AxisConfig.CommandDone;

(* Network 2 *) (* commented out *)
// AxisInterface.Parameters.MovementParameters.Home.EndlessPositionDataRef := pEndlessPosition;

(* Network 3: <axis> Motion Control Function *)
AxisBasic(MpLink := pMpLink, Enable := TRUE, ErrorReset := ErrorReset, Parameters := ADR(AxisInterface.Parameters.MovementParameters), Update := AxisInterface.Commands.ToMapp.Update AND AxisInterface.Status.AxisBasicActive AND NOT AxisBasic.UpdateDone, Axis := pAxis, Power := AxisInterface.Commands.ToMapp.Power, Home := AxisInterface.Commands.ToMapp.Home, MoveVelocity := AxisInterface.Commands.ToMapp.MoveVelocity, MoveAbsolute := AxisInterface.Commands.ToMapp.MoveAbs, MoveAdditive := AxisInterface.Commands.ToMapp.MoveAdditive, Stop := AxisInterface.Commands.ToMapp.Stop, JogPositive := AxisInterface.Commands.ToMapp.JogPos, JogNegative := AxisInterface.Commands.ToMapp.JogNeg, TorqueLimit := AxisInterface.Commands.ToMapp.TorqueLimitingOn);
AxisInterface.Status.AxisBasicActive := AxisBasic.Active;
AxisInterface.Status.Error := AxisBasic.Error;
IF AxisBasic.UpdateDone THEN AxisInterface.Commands.ToMapp.Update := FALSE; END_IF;
AxisInterface.Status.ActualPosition := AxisBasic.Position;
AxisInterface.Status.ActualSpeed := AxisBasic.Velocity;
AxisInterface.Status.MappCommandBusy := AxisBasic.CommandBusy;
AxisInterface.Status.PoweredOn := AxisBasic.PowerOn;
AxisInterface.Status.Homed := AxisBasic.IsHomed;
AxisInterface.Status.InPosition := AxisBasic.InPosition;
AxisInterface.Status.InMotion := AxisBasic.MoveActive;

(* Network 4 *)
AxisInterface.Status.AxisInitialized := AxisBasic.Info.AxisInitialized;
AxisInterface.Status.ReadyToPowerOn := AxisBasic.Info.ReadyToPowerOn;
AxisInterface.Status.ActualTorque := AxisBasic.Info.CyclicRead.Torque.Value;

(* Network 5: The move distance for absolute moves should be the difference between where you are and where you are going *)
_e1(CLK := AxisBasic.MoveAbsolute);
IF _e1.Q THEN
    AbsDistance := ABS(AxisInterface.Parameters.MovementParameters.Position - AxisBasic.Position);
END_IF;

(* Network 6: If the Position Parameter of <axis> has changed, When the move starts add the Calculated distance to the <axis>-Axis Odometer *)
_e2(CLK := AxisBasic.MoveActive);
IF _e2.Q AND AxisBasic.MoveAbsolute THEN OdometerValue := OdometerValue + AbsDistance; END_IF;

(* Network 7 *)
SetOverride(Axis := pAxis, Enable := AxisInterface.Status.PoweredOn, VelFactor := Override, AccFactor := 1.0);
END_FUNCTION_BLOCK
```

### Library Logical/Libraries/Types (IEC)
Depends on: MpAxis

#### Types.typ - Exported data types
```iecst
TYPE
	AdhesCtrlInterface_Commands_typ : 	STRUCT
		MelterOn : BOOL;
		MelterStandbyOff : BOOL;
		MelterStandbyOn : BOOL;
		PumpsOn : BOOL;
		PurgeChannel1 : {REDUND_UNREPLICABLE} BOOL;
		PurgeChannel2 : {REDUND_UNREPLICABLE} BOOL;
		PurgeChannel3 : {REDUND_UNREPLICABLE} BOOL;
		PurgeChannel4 : {REDUND_UNREPLICABLE} BOOL;
		WriteChannelTemp : BOOL;
	END_STRUCT;
	AdhesCtrlInterface_Pars_typ : 	STRUCT
		SavedPatterns : ARRAY[0..3]OF AdhesivePatternCollections_typ;
		AdhesivePatterns : {REDUND_UNREPLICABLE} ARRAY[0..MAX_NUM_GLUE_CHANNELS_M1]OF AdhesivePattern_typ;
		StitchPercentage : {REDUND_UNREPLICABLE} REAL;
		ChannelModulationCtrl : ARRAY[0..MAX_NUM_ONOFF_PATTERNS_M1]OF INT;
		BeadLengths : {REDUND_UNREPLICABLE} ARRAY[0..MAX_NUM_ONOFF_PATTERNS_M1]OF REAL := [4(10)];
		FeedbackIsHardwire : BOOL;
		FeedbackIsModbusTCP : BOOL;
		NordsonComms : NordsonData_typ;
		NordsonFeedbackSelection : NordsonFeedbackSelection_enum;
		NumAdhesiveChannels : {REDUND_UNREPLICABLE} USINT;
		PatternSelection : USINT;
	END_STRUCT;
	AdhesCtrlInterface_Status_typ : 	STRUCT
		AlarmActive : {REDUND_UNREPLICABLE} BOOL;
		ATS_AddOnOverLimit : BOOL;
		ATS_AddOnUnderLimit : BOOL;
		FeederFault : {REDUND_UNREPLICABLE} BOOL;
		GlueApplicationAllowed : {REDUND_UNREPLICABLE} BOOL;
		GlueCyclePos : {REDUND_UNREPLICABLE} REAL;
		LatchedEncoderPos : {REDUND_UNREPLICABLE} REAL;
		LowLevel : {REDUND_UNREPLICABLE} BOOL;
		NordsonInStandby : BOOL;
		ServiceNeeded : {REDUND_UNREPLICABLE} BOOL;
		UnitFault : {REDUND_UNREPLICABLE} BOOL;
		UnitReady : {REDUND_UNREPLICABLE} BOOL;
	END_STRUCT;
	AdhesiveChannelColormaps_typ : 	STRUCT
		Delay : {REDUND_UNREPLICABLE} ARRAY[0..MAX_NUM_ONOFF_PATTERNS_M1]OF USINT;
		Glue : {REDUND_UNREPLICABLE} ARRAY[0..MAX_NUM_ONOFF_PATTERNS_M1]OF USINT;
	END_STRUCT;
	AdhesiveChannelDatapoints_typ : 	STRUCT
		Delay : {REDUND_UNREPLICABLE} ARRAY[0..MAX_NUM_ONOFF_PATTERNS_M1]OF UINT;
		Glue : {REDUND_UNREPLICABLE} ARRAY[0..MAX_NUM_ONOFF_PATTERNS_M1]OF UINT;
		RowLabel : {REDUND_UNREPLICABLE} UINT;
	END_STRUCT;
	AdhesiveCtrlInterface_typ : 	STRUCT
		Commands : {REDUND_UNREPLICABLE} AdhesCtrlInterface_Commands_typ;
		Parameters : {REDUND_UNREPLICABLE} AdhesCtrlInterface_Pars_typ;
		Status : {REDUND_UNREPLICABLE} AdhesCtrlInterface_Status_typ;
	END_STRUCT;
	AdhesivePatternCollections_typ : 	STRUCT
		AdhesivePatterns : ARRAY[0..MAX_NUM_GLUE_CHANNELS_M1]OF AdhesivePattern_typ;
	END_STRUCT;
	AdhesivePattern_typ : 	STRUCT
		DelayDistance : {REDUND_UNREPLICABLE} ARRAY[0..MAX_NUM_ONOFF_PATTERNS_M1]OF REAL;
		GlueOnDistance : {REDUND_UNREPLICABLE} ARRAY[0..MAX_NUM_ONOFF_PATTERNS_M1]OF REAL;
	END_STRUCT;
	AlarmListAdapter_typ : 	STRUCT
		Acknowledged : {REDUND_UNREPLICABLE} ARRAY[0..49]OF STRING[10];
		Active : {REDUND_UNREPLICABLE} ARRAY[0..49]OF STRING[10];
		Code : {REDUND_UNREPLICABLE} ARRAY[0..49]OF STRING[10];
	END_STRUCT;
	AxisInitStates_enum :
		( (*Axis Control States*)
		AXIS_INIT_DONE := 500,
		AXIS_INIT_RETRIEVE_PARS := 10,
		AXIS_INIT_TRANSFER_PARS := 0,
		AXIS_INIT_WAIT_FOR_INIT := 20
		);
	AxisStates_enum :
		( (*Axis Control States*)
		AXIS_STATE_INIT := 0,
		AXIS_STATE_POWERON_PREP := 1,
		AXIS_STATE_POWERON := 2,
		AXIS_STATE_COUPLED := 70,
		AXIS_STATE_ERROR := 999,
		AXIS_STATE_HOME := 30,
		AXIS_STATE_IDLE := 80,
		AXIS_STATE_MOVE := 90,
		AXIS_STATE_MOVE_TO_MASTER := 50,
		AXIS_STATE_MOVE_VELOCITY := 91,
		AXIS_STATE_WAIT_FOR_MASTER_READY := 85,
		AXIS_STATE_W_COUPLE := 60,
		AXIS_STATE_W_HOME := 40
		);
	Axis_enums :
		( (*Axis enumerations*)
		CCW := 4,
		CC_LEFT := 2,
		CC_RIGHT := 3,
		CSW_LEFT := 0,
		CSW_Left11 := 11,
		CSW_Left12 := 12,
		CSW_Left13 := 13,
		CSW_Left14 := 14,
		CSW_Left15 := 15,
		CSW_Left16 := 16,
		CSW_Left17 := 17,
		CSW_Left18 := 18,
		CSW_Left19 := 19,
		CSW_RIGHT := 1,
		FOLDING_ARM_DA_LEFT := 7,
		FOLDING_ARM_DA_RIGHT := 8,
		FOLDING_BAR := 5,
		FOLDING_TOOL_HA_LEFT := 9,
		FOLDING_TOOL_HA_RIGHT := 10,
		FTCL := 6
		);
	Axis_Interface_Comds_ToMapp_typ : 	STRUCT  (*Axis Commands to Mapp*)
		CoupleToMaster : BOOL;
		Home : BOOL;
		JogNeg : BOOL;
		JogPos : BOOL;
		LoadConfig : BOOL;
		MoveAbs : BOOL;
		MoveAdditive : BOOL;
		MoveVelocity : BOOL;
		Power : BOOL;
		SaveConfig : BOOL;
		Stop : BOOL;
		TorqueLimitingOn : BOOL;
		Update : BOOL;
	END_STRUCT;
	Axis_Interface_Commands_typ : 	STRUCT  (*Axis Commands*)
		Init : BOOL;
		MoveVelocityTrigStop : BOOL;
		RequestCoupleToMaster : BOOL;
		RequestHome : BOOL;
		RequestJogNeg : BOOL;
		RequestJogPos : BOOL;
		RequestMoveAbs : BOOL;
		RequestMoveAdditive : BOOL;
		RequestMoveVelocity : BOOL;
		Stop : USINT;
		ToMapp : Axis_Interface_Comds_ToMapp_typ;
	END_STRUCT;
	Axis_Interface_Parameters_typ : 	STRUCT  (*Axis Parameters*)
		AxisAndDrivePars : MpAxisBasicConfigType;
		CouplingMaster : UDINT;
		CouplingParameters : MpAxisCouplingParType;
		MovementParameters : MpAxisBasicParType;
		TriggerDistance : REAL; (*Distance that should be moved after an axis sees a tigger event when using MC_BR_MoveVelocityTriggStop*)
	END_STRUCT;
	Axis_Interface_Status_typ : 	STRUCT  (*Axis Statuses*)
		ActualTorque : LREAL;
		ActualPosition : LREAL;
		ActualSpeed : REAL;
		AxisInitialized : BOOL;
		AxisState : STRING[50];
		ConfigCommandDone : BOOL;
		DefaultRecipeLoaded : BOOL;
		Error : BOOL;
		Homed : BOOL;
		InMotion : BOOL;
		InPosition : BOOL;
		InSync : BOOL;
		MappCommandBusy : BOOL;
		MoveComplete : BOOL;
		PoweredOn : BOOL;
		ReadyToPowerOn : BOOL;
		TriggerMoveDone : BOOL;
		AxisBasicActive : BOOL;
	END_STRUCT;
	Axis_Interface_typ : 	STRUCT  (*servo Axis Interface*)
		Commands : Axis_Interface_Commands_typ;
		Parameters : Axis_Interface_Parameters_typ;
		Status : Axis_Interface_Status_typ;
	END_STRUCT;
	BitmapSelectDatapoints_typ : 	STRUCT
		AlarmActive : {REDUND_UNREPLICABLE} USINT;
		ResetPress : {REDUND_UNREPLICABLE} BOOL;
		RunPress : {REDUND_UNREPLICABLE} BOOL;
		StopPress : {REDUND_UNREPLICABLE} BOOL;
		VacuumPress : {REDUND_UNREPLICABLE} BOOL;
	END_STRUCT;
	Channel_typ : 	STRUCT
		ActualPressure : REAL;
		PressureSetpoint : REAL;
	END_STRUCT;
	ColorMapDatapoints_typ : 	STRUCT
		AdhesiveChannelsColormaps : {REDUND_UNREPLICABLE} ARRAY[0..MAX_NUM_GLUE_CHANNELS_M1]OF AdhesiveChannelColormaps_typ;
		AdhesiveSystemOK : {REDUND_UNREPLICABLE} USINT;
		AdhesiveUnitFault : {REDUND_UNREPLICABLE} USINT;
		AdhesiveUnitFeederFault : {REDUND_UNREPLICABLE} USINT;
		AdhesiveUnitLevelLow : {REDUND_UNREPLICABLE} USINT;
		AdhesiveUnitReady : {REDUND_UNREPLICABLE} USINT;
		AdhesiveUnitServiceNeeded : {REDUND_UNREPLICABLE} USINT;
		AdhesiveUseageLow : {REDUND_UNREPLICABLE} USINT;
		AirPressureOK : {REDUND_UNREPLICABLE} USINT;
		ATSAddOnOver : USINT;
		ATSAddOnUnder : USINT;
		AutoModeSelected : {REDUND_UNREPLICABLE} USINT;
		DownstreamSensorOK : {REDUND_UNREPLICABLE} USINT;
		DriveFaultOK : {REDUND_UNREPLICABLE} USINT;
		GlueSystemOK : {REDUND_UNREPLICABLE} USINT;
		JogModeSelected : {REDUND_UNREPLICABLE} USINT;
		NordsonEditTemps : USINT;
		RecipeLoaded : {REDUND_UNREPLICABLE} USINT;
		RecipeSystemBusy : {REDUND_UNREPLICABLE} USINT;
		SafetyOK : {REDUND_UNREPLICABLE} USINT;
		VacuumOK : {REDUND_UNREPLICABLE} USINT;
		VacuumPressureOK : {REDUND_UNREPLICABLE} USINT;
		VacuumPumpOn : {REDUND_UNREPLICABLE} USINT;
		Valve1OK : {REDUND_UNREPLICABLE} USINT;
		Valve2OK : {REDUND_UNREPLICABLE} USINT;
		Valve3OK : {REDUND_UNREPLICABLE} USINT;
		Valve4OK : USINT;
	END_STRUCT;
	DigitalInputs_typ : 	STRUCT
		AdhesiveLevelLow : {REDUND_UNREPLICABLE} BOOL;
		AdhesivePhotoEye : {REDUND_UNREPLICABLE} BOOL;
		AdhesivePhotoEye_2 : {REDUND_UNREPLICABLE} BOOL;
		AdhesiveUnitNotFaulted : {REDUND_UNREPLICABLE} BOOL;
		AdhesiveUnitReady : {REDUND_UNREPLICABLE} BOOL;
		AirPressureOK : {REDUND_UNREPLICABLE} BOOL;
		BodyDetect : BOOL;
		DownstreamSensor : {REDUND_UNREPLICABLE} BOOL;
		DownstreamSensorRaw : {REDUND_UNREPLICABLE} BOOL;
		LeftEndDetect : BOOL;
		LowAdhesiveUseage : {REDUND_UNREPLICABLE} BOOL;
		Pneumatics580StatusWord3 : {REDUND_UNREPLICABLE} UINT;
		PnuematicsHWStatusV0 : BOOL;
		PnuematicsHWStatusV2 : BOOL;
		PnuematicsHWStatusV4 : BOOL;
		PnuematicsHWStatusV6 : BOOL;
		RightEndDetect : BOOL;
		SafetyOK : {REDUND_UNREPLICABLE} BOOL;
		SSI_Parallel : {REDUND_UNREPLICABLE} SSI_Paraller_typ;
		VacHigh : BOOL;
		VacLow : BOOL;
		VacuumPressureOK : {REDUND_UNREPLICABLE} BOOL;
		VacuumTempOK : {REDUND_UNREPLICABLE} BOOL;
		X_PickRetracted : BOOL;
		X_PickExtended : BOOL;
		Y_PickRetract : BOOL;
		X_BlowOff : BOOL;
		BodyHopperLow : BOOL;
		HopperMotor_RUN : BOOL;
		LubricationCounter : BOOL;
		HopperMotor_OFF : BOOL;
		DownstreamSensorON : BOOL;
	END_STRUCT;
	DigitalOutputs_typ : 	STRUCT
		AirOn : {REDUND_UNREPLICABLE} BOOL;
		AmberLightStack : {REDUND_UNREPLICABLE} BOOL;
		BlowOffOn : BOOL;
		BottomFolder : {REDUND_UNREPLICABLE} BOOL;
		CompressionAirOn : BOOL;
		GlueChannel1 : {REDUND_UNREPLICABLE} BOOL;
		GlueChannel2 : {REDUND_UNREPLICABLE} BOOL;
		GlueChannel3 : {REDUND_UNREPLICABLE} BOOL;
		GlueChannel4 : {REDUND_UNREPLICABLE} BOOL;
		GreenLightStack : {REDUND_UNREPLICABLE} BOOL;
		HighCompression : BOOL;
		LowCompression : BOOL;
		PickAndPlace_X : BOOL;
		Pneumatics580ControlWord1 : {REDUND_UNREPLICABLE} UINT;
		PnuematicsValve0 : BOOL;
		PnuematicsValve2 : BOOL;
		PnuematicsValve4 : BOOL;
		PnuematicsValve6 : BOOL;
		PushOn : {REDUND_UNREPLICABLE} BOOL;
		RedLightStack : {REDUND_UNREPLICABLE} BOOL;
		ResetEuchner : BOOL;
		ResetSafety : {REDUND_UNREPLICABLE} BOOL;
		TopFolder : {REDUND_UNREPLICABLE} BOOL;
		VacuumOn : {REDUND_UNREPLICABLE} BOOL;
		ZeroEncoder : {REDUND_UNREPLICABLE} BOOL;
		SidePanelVacOn : BOOL;
		SidePanelVacBlowOff : BOOL;
		X_PickSolenoid : BOOL;
		Y_PickSolenoid : BOOL;
	END_STRUCT;
	Encoders_typ : {REDUND_UNREPLICABLE} 	STRUCT
		SickSSIPos : {REDUND_UNREPLICABLE} UDINT;
		SickSSIPosDegrees : {REDUND_UNREPLICABLE} REAL;
		FeedEncoderPos : {REDUND_UNREPLICABLE} UDINT;
		FeedEncoderPosDegrees : {REDUND_UNREPLICABLE} REAL;
		RamEncoderPos : {REDUND_UNREPLICABLE} UDINT;
		RamEncoderPosDegrees : {REDUND_UNREPLICABLE} REAL;
	END_STRUCT;
	FolderTypeSelection_enum :
		(
		FOLDER_LINMOT := 1,
		FOLDER_PNEUMATIC := 0
		);
	FoldpushCtrlInterface_Pars_typ : 	STRUCT
		BottomFolderOffPos : REAL;
		BottomFolderOnPos : REAL;
		FolderTypeSelection : FolderTypeSelection_enum;
		HighCompressionOffPos : REAL;
		HighCompressionOnPos : REAL;
		LinMotBotFolder : LinAxis_typ;
		LinMotTopFolder : LinAxis_typ;
		LowCompressionOffPos : REAL;
		LowCompressionOnPos : REAL;
		NumaticsTypeSelection : NumaticsTypeSelection_enum;
		PushOff : {REDUND_UNREPLICABLE} REAL;
		PushOn : {REDUND_UNREPLICABLE} REAL;
		TopFolderOffPos : REAL;
		TopFolderOnPos : REAL;
	END_STRUCT;
	FoldpushCtrlInterface_Status_typ : 	STRUCT
		BottomFoldValveStatus : {REDUND_UNREPLICABLE} BOOL;
		CompOnValveStatus : BOOL;
		CompressionAllowed : BOOL;
		FoldersActuationAllowed : {REDUND_UNREPLICABLE} BOOL;
		HardwireConfig : BOOL;
		LinMotConfig : BOOL;
		PneumaticConfig : BOOL;
		PowelinkConfig : BOOL;
		PushValveStatus : {REDUND_UNREPLICABLE} BOOL;
		TopFoldValveStatus : {REDUND_UNREPLICABLE} BOOL;
	END_STRUCT;
	FoldPushCtrlInterface_typ : 	STRUCT
		Commands : {REDUND_UNREPLICABLE} FoldPushCtrlInt_Commands_typ;
		Parameters : {REDUND_UNREPLICABLE} FoldpushCtrlInterface_Pars_typ;
		Status : {REDUND_UNREPLICABLE} FoldpushCtrlInterface_Status_typ;
	END_STRUCT;
	FoldPushCtrlInt_Commands_typ : 	STRUCT
		placehold : {REDUND_UNREPLICABLE} BOOL;
	END_STRUCT;
	HMIControl_Commands_typ : 	STRUCT
		CancelBoxChange : BOOL;
		ConfirmBoxChange : BOOL;
		CycleServoHopper : BOOL;
		CycleServoRam : BOOL;
		HomeServoFeed : BOOL;
		HomeServoHopper : BOOL;
		HomeServoRam : BOOL;
		JogForward : BOOL;
		JogReverse : BOOL;
		JogServoFeedNeg : BOOL;
		JogServoFeedPos : BOOL;
		JogServoHopperNeg : BOOL;
		JogServoHopperPos : BOOL;
		JogServoRamNeg : BOOL;
		JogServoRamPos : BOOL;
		LoadRecipe : BOOL;
		LoadRecipeType1 : BOOL;
		LoadRecipeType2 : BOOL;
		RequestBoxType1 : BOOL;
		RequestBoxType2 : BOOL;
		RequestReset : BOOL;
		RequestStop : BOOL;
		RequestVacuumOn : BOOL;
		RequestVFDRun : BOOL;
		SaveRecipe : BOOL;
		SelectAutoMode : BOOL;
		SelectJogMode : BOOL;
		StartServoFeed : BOOL;
		StartServoHopper : BOOL;
		ZeroEncoder : BOOL;
		EnableShowMode : BOOL;
	END_STRUCT;
	HMIControl_Parameters_typ : 	STRUCT
		ServoFeedAccel : REAL;
		ServoFeedJogVelocity : REAL;
		ServoFeedTorqueLimit : REAL;
		ServoFeedVelocity : REAL;
		ServoHopperAccel : REAL;
		ServoHopperEndDwellTime : UDINT;
		ServoHopperEndPosition : REAL;
		ServoHopperJogVelocity : REAL;
		ServoHopperStartDwellTime : UDINT;
		ServoHopperStartPosition : REAL;
		ServoHopperTorqueLimit : REAL;
		ServoHopperVelocity : REAL;
		ServoRamAccel : REAL;
		ServoRamEndDwellTime : UDINT;
		ServoRamEndPosition : REAL;
		ServoRamJogVelocity : REAL;
		ServoRamStartDwellTime : UDINT;
		ServoRamStartPosition : REAL;
		ServoRamTorqueLimit : REAL;
		ServoRamNegativeVelocity : REAL;
		ServoRamPositiveVelocity : REAL;
		ServoRamClearPosition : REAL;
		PickAndPlaceDwell : UDINT;
		ServoHopperDwellTime : UDINT;
		AtTorqueTime : UDINT;
		PickDwellTime : UDINT;
		TopFeedJamTime : UDINT;
		VacuumOffTime : UDINT;
		DownPulseTime : UDINT;
		Y_DelayTime : UDINT;
		BlowOffTime : UDINT;
		SetCycleCount : UDINT;
		LubeCycleCount : UDINT;
		LowFeedJamTime : UDINT;
		LowHopperTime : UDINT;
	END_STRUCT;
	HMIControl_typ : 	STRUCT
		BitmapSelectDatapoints : {REDUND_UNREPLICABLE} BitmapSelectDatapoints_typ;
		ColorMapDatapoints : {REDUND_UNREPLICABLE} ColorMapDatapoints_typ;
		Commands : {REDUND_UNREPLICABLE} HMIControl_Commands_typ;
		Parameters : HMIControl_Parameters_typ;
		StatusDatapoints : {REDUND_UNREPLICABLE} StatusDatapoints_typ;
	END_STRUCT;
	Home_Parameters_typ : 	STRUCT  (*Axis Homing Parameters*)
		ServoFeed : MpAxisHomingType;
		ServoHopper : MpAxisHomingType;
		ServoRam : MpAxisHomingType;
	END_STRUCT;
	IO_typ : 	STRUCT
		DIs : {REDUND_UNREPLICABLE} DigitalInputs_typ;
		DOs : {REDUND_UNREPLICABLE} DigitalOutputs_typ;
		Encoders : {REDUND_UNREPLICABLE} Encoders_typ;
		ModuleOKs : {REDUND_UNREPLICABLE} ARRAY[0..99]OF BOOL;
		SafetyStatus : SafetyStatus_typ;
	END_STRUCT;
	LightStack_typ :
		(
		LIGHTSTACK_PATLITE := 1,
		LIGHTSTACK_TRI := 0
		);
	LinAxisCommand_typ : 	STRUCT  (*Axis command type*)
		ErrorReset : BOOL; (*Reset error command*)
		Home : BOOL; (*Home command*)
		HomeRequest : BOOL; (*Request for home from HMI*)
		JogNegative : BOOL; (*Jog neg command*)
		JogNegativeRequest : BOOL; (*Request for jog negative*)
		JogPositive : BOOL; (*Jog pos command*)
		JogPositiveRequest : BOOL; (*Request for jog positive*)
		MoveAbsolute : BOOL; (*Move absolute command*)
		MoveAbsoluteRequest : BOOL; (*Request for move absolute*)
		MoveAdditive : BOOL; (*Move additive command*)
		Power : BOOL; (*Power command*)
		SaveConfig : BOOL;
		Stop : BOOL; (*Stop command*)
	END_STRUCT;
	LinAxisParameter_typ : 	STRUCT  (*Axis parameter type*)
		ExtendAccel : REAL;
		ExtendDecel : REAL;
		ExtendPos : LREAL;
		ExtendSpeed : REAL;
		MpBasicConfig : MpAxisBasicConfigType; (*Axis configuration parameters for change at runtime*)
		MpBasicParameters : MpAxisBasicParType; (*Mp params*)
		RetractAccel : REAL;
		RetractDecel : REAL;
		RetractPos : LREAL;
		RetractSpeed : REAL;
	END_STRUCT;
	LinAxisStatus_typ : 	STRUCT  (*Axis status type*)
		EndlessPosValid : BOOL; (*Endless position is valid*)
		Error : BOOL; (*Error active on axis*)
		ErrorId : DINT; (*Error id*)
		HomeCheck : BOOL;
		Info : MpAxisBasicInfoType;
		InPosition : BOOL; (*Axis in position*)
		IsHomed : BOOL; (*Axis is homed*)
		MoveActive : BOOL; (*Move is active on the axis*)
		Position : LREAL; (*Current position of axis*)
		PowerOn : BOOL; (*Axis is on*)
		Ready : BOOL; (*Axis is in standstill and homed*)
		Stopped : BOOL; (*Axis is stopped*)
		Velocity : REAL; (*Current velocity of axis*)
	END_STRUCT;
	LinAxis_typ : 	STRUCT  (*Axis type*)
		Command : LinAxisCommand_typ; (*Command*)
		Parameter : LinAxisParameter_typ; (*Parameter*)
		Status : LinAxisStatus_typ; (*Status*)
	END_STRUCT;
	LinMotState_enum :
		(
		STATE_ERROR,
		STATE_HOME_CHECK,
		STATE_HOME_RESTORE,
		STATE_HOME_STANDBY,
		STATE_HOME_TORQUE,
		STATE_INIT,
		STATE_IS_HOMED,
		STATE_JOG_NEG,
		STATE_JOG_POS,
		STATE_MOVE,
		STATE_READY
		);
	ModeCtrlInterface_Commands_typ : {REDUND_UNREPLICABLE} 	STRUCT
		FinishCycle : {REDUND_UNREPLICABLE} BOOL;
		ForceSafetyReset : {REDUND_UNREPLICABLE} BOOL;
		Reset : {REDUND_UNREPLICABLE} BOOL;
		Run : {REDUND_UNREPLICABLE} BOOL;
		SetAutoMode : {REDUND_UNREPLICABLE} BOOL;
		SetJogMode : {REDUND_UNREPLICABLE} BOOL;
		Stop : {REDUND_UNREPLICABLE} BOOL;
		SetShowMode : {REDUND_UNREPLICABLE} BOOL;
	END_STRUCT;
	ModeCtrlInterface_Parameters_typ : 	STRUCT
		BottomSensor : BOOL;
		DownstreamClear : UDINT := 1000;
		DownstreamIgnored : BOOL;
		DownstreamTimeout : UDINT := 1000;
		DwellTime : {REDUND_UNREPLICABLE} UDINT;
		InPositionTolerance : REAL := 10.0;
		LightStackSelection : LightStack_typ;
		MachineType : USINT;
		MaxPPM : UINT;
		MinPPM : UINT;
		PiecesPerMinute : {REDUND_UNREPLICABLE} UINT;
		SideSensors : BOOL;
		StopPosition : {REDUND_UNREPLICABLE} REAL;
		VaccumStopTime : UDINT := 200;
	END_STRUCT;
	ModeCtrlInterface_Status_typ : 	STRUCT
		AtStopPosition : {REDUND_UNREPLICABLE} BOOL;
		BlissPanelAlarmActive : BOOL;
		Dwelling : {REDUND_UNREPLICABLE} BOOL;
		DwellModeEnabled : {REDUND_UNREPLICABLE} BOOL;
		InAutoMode : {REDUND_UNREPLICABLE} BOOL;
		InBlissPanelWindow : BOOL;
		Jogging : {REDUND_UNREPLICABLE} BOOL;
		MachineIsBliss : BOOL;
		Running : {REDUND_UNREPLICABLE} BOOL;
		WaitingOnDownstream : BOOL;
	END_STRUCT;
	ModeCtrlInterface_typ : 	STRUCT
		Commands : {REDUND_UNREPLICABLE} ModeCtrlInterface_Commands_typ;
		Parameters : {REDUND_UNREPLICABLE} ModeCtrlInterface_Parameters_typ;
		Status : ModeCtrlInterface_Status_typ;
	END_STRUCT;
	NordsonData_typ : 	STRUCT
		AdhesiveUsePerHour : UDINT;
		Alert : BOOL;
		ByPassFeedback : BOOL;
		ChannelActTemp : ARRAY[0..NUM_NORDSON_TEMP_ZONES_M1]OF UINT;
		ChannelDataCmpResult : DINT;
		ChannelDataSize : UDINT;
		ChannelSetTempActual : ARRAY[0..NUM_NORDSON_TEMP_ZONES_M1]OF UINT;
		ChannelSetTempRequested : ARRAY[0..NUM_NORDSON_TEMP_ZONES_M1]OF UINT;
		CommFault : BOOL;
		CommFaultInDataValue : BOOL;
		ConsecutiveErrorCount : USINT;
		FeedbackTime : TIME := T#1s;
		HeatUpPhaseActive : BOOL;
		HoseSetTemp : UINT;
		MelterIsOn : BOOL;
		MelterStatus : UINT;
		PumpStartUpProtectionOn : BOOL;
		ShutDown : BOOL;
		StandbyTimeoutTime : TIME := T#2h;
		TempUnit : USINT;
		UnitFaulted : BOOL;
		UnitReady : BOOL;
	END_STRUCT;
	NordsonFeedbackSelection_enum :
		(
		NORDSON_HARDWIRE := 0,
		NORDSON_MODBUSTCP := 1
		);
	NordsonRxPacket_typ : 	STRUCT
		Byte0_1_Status : UINT;
		Byte2_Ack_Data_Index : USINT;
		Byte3_Ack_Channel_Num : USINT;
		Byte4_5_Read_Data_0 : UINT;
		Byte6_7_Read_Data_1 : UINT;
		Byte8_9_Read_Data_2 : UINT;
		Byte10_11_Read_Data_3 : UINT;
		Byte12_13_Read_Data_4 : UINT;
		Byte14_15_Read_Data_5 : UINT;
	END_STRUCT;
	NordsonTxPacket_typ : 	STRUCT
		Byte0_MelterControl : USINT;
		Byte1_Command : USINT;
		Byte2_Data_Index : USINT;
		Byte3_Channel_Num : USINT;
		Byte4_5_WriteData : UINT;
		Byte6_7_Mot1Spd : UINT;
		Byte8_9_Mot2Spd : UINT;
		Byte10_11_Mot3Spd : UINT;
		Byte12_13_Mot4Spd : UINT;
		Byte14_15_NotUsed : UINT;
	END_STRUCT;
	NumaticsTypeSelection_enum :
		(
		NUMATICS_HARDWIRE,
		NUMATICS_POWERLINK
		);
	RamControlInterface_typ : 	STRUCT
		Commands : {REDUND_UNREPLICABLE} RamCtrlInterface_Commands_typ;
		Parameters : {REDUND_UNREPLICABLE} RamCtrlInterface_Parameters_typ;
		Status : {REDUND_UNREPLICABLE} RamCtrlInterface_Status_typ;
	END_STRUCT;
	RamCtrlInterface_Commands_typ : 	STRUCT
		Home : {REDUND_UNREPLICABLE} BOOL;
		JogNegative : {REDUND_UNREPLICABLE} BOOL;
		JogPositive : {REDUND_UNREPLICABLE} BOOL;
		MoveAbsolute : {REDUND_UNREPLICABLE} BOOL;
		MoveAdditive : {REDUND_UNREPLICABLE} BOOL;
		MoveVelocity : {REDUND_UNREPLICABLE} BOOL;
		PowerOn : {REDUND_UNREPLICABLE} BOOL;
		VFDAlarmReset : {REDUND_UNREPLICABLE} BOOL;
	END_STRUCT;
	RamCtrlInterface_Parameters_typ : 	STRUCT
		Acceleration : {REDUND_UNREPLICABLE} REAL;
		CurrentLimit : {REDUND_UNREPLICABLE} REAL;
		GearRatio : REAL := 54;
		JogSpeed : {REDUND_UNREPLICABLE} REAL;
		Position : {REDUND_UNREPLICABLE} REAL;
	END_STRUCT;
	RamCtrlInterface_Status_typ : 	STRUCT
		ActualPosition : {REDUND_UNREPLICABLE} LREAL;
		ActualSpeed : {REDUND_UNREPLICABLE} LREAL;
		AlarmActive : {REDUND_UNREPLICABLE} BOOL;
		DriveSpeed : {REDUND_UNREPLICABLE} INT;
		Home : {REDUND_UNREPLICABLE} BOOL;
		InPosition : {REDUND_UNREPLICABLE} BOOL;
		MotorCurrent : {REDUND_UNREPLICABLE} UINT;
		MoveActive : {REDUND_UNREPLICABLE} BOOL;
		Position : {REDUND_UNREPLICABLE} REAL;
		PoweredOn : {REDUND_UNREPLICABLE} BOOL;
		Running : {REDUND_UNREPLICABLE} BOOL;
		Stopped : BOOL;
		STOStatus : UINT;
		VFDAlarmDetected : {REDUND_UNREPLICABLE} BOOL;
		VFDAlarmNumber : {REDUND_UNREPLICABLE} INT;
		VFDAlarmText : {REDUND_UNREPLICABLE} STRING[80];
	END_STRUCT;
	RecipeCtrlInterface_Commands_typ : 	STRUCT
		ChangeRecipe : BOOL;
		LoadRecipe : {REDUND_UNREPLICABLE} BOOL;
		SaveRecipe : {REDUND_UNREPLICABLE} BOOL;
	END_STRUCT;
	RecipeCtrlInterface_Pars_typ : 	STRUCT
		RecipeIndex : USINT;
		RecipeName : {REDUND_UNREPLICABLE} STRING[100];
	END_STRUCT;
	RecipeCtrlInterface_Status_typ : 	STRUCT
		Busy : {REDUND_UNREPLICABLE} BOOL;
		LoadedRecipeIndex : USINT;
		LoadedRecipeName : {REDUND_UNREPLICABLE} STRING[255];
		RecipeHasBeenLoaded : BOOL;
	END_STRUCT;
	RecipeCtrlInterface_typ : 	STRUCT
		Commands : {REDUND_UNREPLICABLE} RecipeCtrlInterface_Commands_typ;
		Parameters : {REDUND_UNREPLICABLE} RecipeCtrlInterface_Pars_typ;
		Status : {REDUND_UNREPLICABLE} RecipeCtrlInterface_Status_typ;
	END_STRUCT;
	Register_typ : 	STRUCT
		ChannelActualPressureWord : UDINT;
		ChannelSetPressureWord : UDINT;
		TankActualLevelWord : UINT;
	END_STRUCT;
	SafetyStatus_typ : 	STRUCT
		BackEstopOK : BOOL;
		CabinetEStopStatus : UINT;
		FrontEStopOK : BOOL;
		GuardDoorsOK : BOOL;
		SafetyProgramRunning : BOOL;
	END_STRUCT;
	SSI_Paraller_typ : {REDUND_UNREPLICABLE} 	STRUCT
		Bits : {REDUND_UNREPLICABLE} ARRAY[0..15]OF BOOL;
		FeedBits : {REDUND_UNREPLICABLE} ARRAY[0..15]OF BOOL;
		RamBits : {REDUND_UNREPLICABLE} ARRAY[0..15]OF BOOL;
	END_STRUCT;
	StatusDatapoints_typ : 	STRUCT
		AdhesiveChannelSDPs : {REDUND_UNREPLICABLE} ARRAY[0..MAX_NUM_GLUE_CHANNELS_M1]OF AdhesiveChannelDatapoints_typ;
		AdhesivePatternDialogSDP : UINT := 1;
		AdhesivePatternConfirmDialogSDP : UINT := 1;
		AdhesivePatternConfirmedSDP : UINT;
		AdhesiveUnitFaultSDP : {REDUND_UNREPLICABLE} UINT;
		AdhesiveUnitLevelLowSDP : {REDUND_UNREPLICABLE} UINT;
		AdhesiveUnitNotReadySDP : {REDUND_UNREPLICABLE} UINT;
		AdhesiveUseageLowSDP : {REDUND_UNREPLICABLE} UINT;
		AutoModeSDP : {REDUND_UNREPLICABLE} UINT;
		BlissSDP : UINT;
		HardwireValveSDP : USINT;
		JogStatusDatapoint : {REDUND_UNREPLICABLE} UINT;
		LinMotBotHomeSDP : UINT;
		LinMotSDP : UINT;
		LinMotTopHomeSDP : UINT;
		LinMotTuningSDP : UINT;
		MaintenanceSDP : {REDUND_UNREPLICABLE} UINT;
		MotorVacuumSDP : UINT;
		NordsonModbusSDP : UINT;
		NordsonStandbyOffSDP : UINT;
		PnuematicFolderSDP : UINT;
		RecipeDialogSDP : UINT;
		RecipeIndexSDP : UINT;
		RecipeReq1SDP : UINT;
		RecipeReq2SDP : UINT;
		RestartInhibitSDP : UINT;
		SafetyStartingSDP : UINT;
		ServoLayerSDP : {REDUND_UNREPLICABLE} UINT;
		ServoRamHomeSDP : UINT;
		SmartVacuumLayerSDP : {REDUND_UNREPLICABLE} UINT;
		TraySDP : UINT;
		VacuumPressureFaultSDP : {REDUND_UNREPLICABLE} UINT;
		VenturiVacuumSDP : UINT;
		ZeroEncoderSDP : {REDUND_UNREPLICABLE} UINT;
		HopperLowSDP : UINT;
		HomeServoRamSDP : UINT;
		LubeSDP : UINT;
	END_STRUCT;
	Tank_typ : 	STRUCT
		ActualLevel : REAL;
	END_STRUCT;
	VacCtrlConfig_enum :
		(
		VAC_MOTOR := 0,
		VAC_VENTURI := 1
		);
	VacCtrlInterface_Commands_typ : 	STRUCT
		BlowOffOnManual : BOOL;
		VacuumOn : {REDUND_UNREPLICABLE} BOOL;
		VenturiOn : BOOL;
		VenturiOnManual : BOOL;
	END_STRUCT;
	VacCtrlInterface_Parameters_typ : 	STRUCT
		BlowOffTime : UINT;
		ManualVenturiVacuumOff : BOOL;
		VacConfig : VacCtrlConfig_enum;
		VacOffPos : REAL;
		VacOnPos : REAL;
	END_STRUCT;
	VacCtrlInterface_Status_typ : 	STRUCT
		AlarmActive : {REDUND_UNREPLICABLE} BOOL;
		Pressure : {REDUND_UNREPLICABLE} REAL;
		StandstillTimout : BOOL;
		StandstillTimoutSet : BOOL;
		VacLowAlarm : BOOL;
		VacLowCycle : BOOL;
	END_STRUCT;
	VacCtrlInterface_typ : 	STRUCT
		Commands : {REDUND_UNREPLICABLE} VacCtrlInterface_Commands_typ;
		Parameters : {REDUND_UNREPLICABLE} VacCtrlInterface_Parameters_typ;
		Status : {REDUND_UNREPLICABLE} VacCtrlInterface_Status_typ;
	END_STRUCT;
END_TYPE
```

### Library Logical/Libraries/AxisFUBs (ANSIC)
Depends on: Types, standard

#### AxisFUBs.fun - Exported functions and function blocks
```iecst
{REDUND_ERROR} FUNCTION_BLOCK AxisHandler (*Implements state machine for single axis handling*) (*$GROUP=User,$CAT=User,$GROUPICON=User.png,$CATICON=User.png*)
	VAR_INPUT
		FirstHomeExecuted : REFERENCE TO BOOL;
		pInterface : REFERENCE TO Axis_Interface_typ;
		pHomingParameters : REFERENCE TO MpAxisHomingType;
		AlarmActive : BOOL;
		IsSimulated : BOOL;
	END_VAR
	VAR
		state : AxisStates_enum := 0;
		axisInitState : AxisInitStates_enum;
		DriveReadyTimeout : TON;
		SetOverride : MC_SetOverride;
	END_VAR
END_FUNCTION_BLOCK
```

#### AxisHandler.c
```c
#include <bur/plctypes.h>
#include "string.h"

#ifdef __cplusplus
	extern "C"
	{
#endif
#include "AxisFUBs.h"
#ifdef __cplusplus
	};
#endif
/* Implements state machine for single axis handling */
void AxisHandler(struct AxisHandler* t)
{

	if(t->AlarmActive == 1) {
		t->state = AXIS_STATE_ERROR;
	}

	//force these off. State machine will set them if jog is requested and state allows it
	t->pInterface->Commands.ToMapp.JogNeg = 0;
	t->pInterface->Commands.ToMapp.JogPos = 0;
	t->pInterface->Parameters.MovementParameters.Deceleration = t->pInterface->Parameters.MovementParameters.Acceleration;

	t->pInterface->Parameters.MovementParameters.Jog.LowerLimit = 0;

	t->DriveReadyTimeout.IN = 0; //will be set true in appropriate state(s)

	//	switch (t->axisInitState){
	//		//init the axis/drive
	//		case AXIS_INIT_TRANSFER_PARS:
	//
	//		//	strcpy((char*)&t->pInterface->Status.AxisState, "Loading Axis Parameters");
	//
	//		//	if(t->pSystemInterface->Status.DefaultRecipeLoaded == 1) //axis parameters should be part of the recipe system and are only 'good' once recipe system has loaded the values
	//			if(1)
	//			{
	//				//unclear if axis parameters will become part of the recipe system, so just continue on for now - jdl
	////				t->pInterface->Commands.ToMapp.SaveConfig = 1;
	////
	////				if(t->pInterface->Status.ConfigCommandDone){
	////					t->pInterface->Commands.ToMapp.SaveConfig = 0;
	////				}
	//
	//				t->axisInitState = AXIS_INIT_RETRIEVE_PARS;
	//			}
	//			break;
	//
	//		//Get mapp config parameters. These should ideally come from the recipe system
	//		case AXIS_INIT_RETRIEVE_PARS:
	//
	//		//	strcpy((char*)&t->pInterface->Status.AxisState, "Retrieving Axis Parameters");
	//
	//			t->pInterface->Commands.ToMapp.LoadConfig = 1;
	//
	//			if(t->pInterface->Status.ConfigCommandDone){
	//				t->pInterface->Commands.ToMapp.LoadConfig = 0;
	//				t->axisInitState = AXIS_INIT_WAIT_FOR_INIT;
	//			}
	//			break;
	//
	//		//Get mapp config parameters. These should ideally come from the recipe system
	//		case AXIS_INIT_WAIT_FOR_INIT:
	//
	//			//	strcpy((char*)&t->pInterface->Status.AxisState, "Retrieving Axis Parameters");
	//
	//			t->pInterface->Commands.ToMapp.Update = 1;
	//
	//			if(t->pInterface->Status.AxisInitialized){
	//				t->axisInitState = AXIS_INIT_DONE;
	//			}
	//			break;
	//
	//		case AXIS_INIT_DONE:
	//			if(t->pInterface->Commands.Init){
	//				t->pInterface->Commands.Init = 0;
	//				t->axisInitState = AXIS_INIT_TRANSFER_PARS;
	//			}
	//	}

	switch (t->state)
	{
		case AXIS_STATE_INIT:

			if (t->pInterface->Status.AxisBasicActive) {

				//force parameter save to the drive. values are set in init code of motion handler
				t->pInterface->Commands.ToMapp.SaveConfig = 1;

				if(t->pInterface->Status.ConfigCommandDone){
					t->pInterface->Commands.ToMapp.SaveConfig = 0;
					t->pInterface->Commands.ToMapp.Update = 0;
				}
				t->state = AXIS_STATE_POWERON_PREP;
			}
			break;

		//we need at least one scan where the power on command is 0. handles cases where the power on command is always true and the machine can't power on.
		case AXIS_STATE_POWERON_PREP:

			t->pInterface->Commands.ToMapp.Update = 1;

			if (t->pInterface->Status.AxisInitialized) {
				t->pInterface->Commands.ToMapp.Power = 0;
				t->state = AXIS_STATE_POWERON;
			}
			break;

		//power on the Drive
		case AXIS_STATE_POWERON:

			strcpy((char*)&t->pInterface->Status.AxisState, "Powering On");
			t->DriveReadyTimeout.IN = 1; //will be cleared outside of state machine

			if ((t->pInterface->Status.ReadyToPowerOn) || (t->DriveReadyTimeout.Q))  //Issue the power on command if drives do not become ready with in time out.  The drive will then post an alarm to explain why it won't power on.
			{
				t->DriveReadyTimeout.IN = 0;
				t->pInterface->Commands.ToMapp.Power = 1;

				if(t->pInterface->Status.PoweredOn)
				{
					t->state = AXIS_STATE_HOME;
				}
			}
			break;

		//On start up, home the axis
		case AXIS_STATE_HOME:

			strcpy((char*)&t->pInterface->Status.AxisState, "Waiting To Start Home");

			if(t->pInterface->Status.ReadyToPowerOn == 1)
			{
				if((*t->FirstHomeExecuted == 0) || (!t->pInterface->Status.Homed))
				{
					//if system is simulated or the home mode is direct home, just direct home
					if((t->IsSimulated) || (t->pHomingParameters->Mode == mpAXIS_HOME_MODE_DIRECT)) {
					//if(t->IsSimulated) {
					t->pInterface->Parameters.MovementParameters.Home.Position = 0;
					t->pInterface->Parameters.MovementParameters.Home.SensorOffset = 0;
					t->pInterface->Parameters.MovementParameters.Home.Mode = mpAXIS_HOME_MODE_DIRECT;

					t->pInterface->Commands.RequestHome = 0;
					t->pInterface->Commands.ToMapp.Home = 1;
					t->state = AXIS_STATE_W_HOME;
					}
					else if(t->pInterface->Commands.RequestHome) //Otherwise execute set home routine
					{
					memcpy(&t->pInterface->Parameters.MovementParameters.Home, t->pHomingParameters, sizeof(t->pInterface->Parameters.MovementParameters.Home));

					t->pInterface->Commands.RequestHome = 0;
					t->pInterface->Commands.ToMapp.Home = 1;
					t->state = AXIS_STATE_W_HOME;
					}
				}
					//				else if(!t->pInterface->Status.Homed) //got to this state with a good stored position but we aren't homed, so recall the position
					//				{
					//					t->pInterface->Parameters.MovementParameters.Home.SensorOffset = 0;
					//					t->pInterface->Parameters.MovementParameters.Home.Mode = mpAXIS_HOME_MODE_RESTORE_POS;
					//					t->pInterface->Commands.ToMapp.Home = 1;
					//					t->state = AXIS_STATE_W_HOME;
					//				}
				else if(t->pInterface->Status.Homed) //got to this state without requesting home, and we're already homed. Probably recovering from error, just go to idle
				{
					t->state = AXIS_STATE_IDLE;
				}
			}
			break;

		// wait for home to finish
		case AXIS_STATE_W_HOME:

			strcpy((char*)&t->pInterface->Status.AxisState, "Homing");

			if(t->pInterface->Status.Homed)
			{
				t->pInterface->Commands.ToMapp.Home = 0;
				*t->FirstHomeExecuted = 1; //a home has been completed successfully, we do not need the home routine again
				t->state = AXIS_STATE_IDLE;
			}
			break;

		//Idle state. Ready to receive commands for commands
		case AXIS_STATE_IDLE:

			strcpy((char*)&t->pInterface->Status.AxisState, "Idle");

			if(t->pInterface->Commands.RequestHome == 1)
			{
				*t->FirstHomeExecuted = 0;
				t->state = AXIS_STATE_HOME;
			}
			else if(t->pInterface->Commands.RequestMoveAbs == 1)
			{
				t->pInterface->Commands.RequestMoveAbs = 0;
				t->pInterface->Commands.ToMapp.MoveAbs = 1;
				t->state = AXIS_STATE_MOVE;
			}
			else if(t->pInterface->Commands.RequestMoveAdditive == 1)
			{
				t->pInterface->Commands.RequestMoveAdditive = 0;
				t->pInterface->Commands.ToMapp.MoveAdditive = 1;
				t->state = AXIS_STATE_MOVE;
			}
			else if(t->pInterface->Commands.RequestMoveVelocity == 1)
			{
				t->pInterface->Commands.ToMapp.MoveVelocity = 1;
				t->state = AXIS_STATE_MOVE_VELOCITY;
			}
			else if(t->pInterface->Commands.RequestJogNeg)
			{
				t->pInterface->Commands.ToMapp.JogNeg = 1;
			}
			else if(t->pInterface->Commands.RequestJogPos)
			{
				t->pInterface->Commands.ToMapp.JogPos = 1;
			}
			else if(t->pInterface->Commands.RequestCoupleToMaster)
			{
				t->pInterface->Commands.ToMapp.CoupleToMaster = 1;
				t->state = AXIS_STATE_W_COUPLE;
			}
			break;

		case AXIS_STATE_MOVE:

			strcpy((char*)&t->pInterface->Status.AxisState, "In Motion");

			if((t->pInterface->Status.InPosition == 1) && (t->pInterface->Status.MappCommandBusy == 0)){
				t->pInterface->Status.MoveComplete = 1;
				t->pInterface->Commands.ToMapp.MoveAbs = 0;
				t->pInterface->Commands.ToMapp.MoveAdditive = 0;
				t->state = AXIS_STATE_IDLE;
			}
			break;

		case AXIS_STATE_MOVE_VELOCITY:

			strcpy((char*)&t->pInterface->Status.AxisState, "In Velocity");

			if(t->pInterface->Commands.RequestMoveVelocity == 0){
				t->pInterface->Commands.ToMapp.MoveVelocity = 0;
				t->state = AXIS_STATE_IDLE;
			}

			break;

		case AXIS_STATE_W_COUPLE:

			strcpy((char*)&t->pInterface->Status.AxisState, "Waiting To Couple To Master");

			if(t->pInterface->Status.InSync){
				t->state = AXIS_STATE_COUPLED;
			}

			break;

		case AXIS_STATE_COUPLED:

			strcpy((char*)&t->pInterface->Status.AxisState, "Coupled To Master");

			if(!(t->pInterface->Commands.RequestCoupleToMaster)){
				t->pInterface->Commands.ToMapp.CoupleToMaster = 0;

				if(!(t->pInterface->Status.InSync)){
					t->state = AXIS_STATE_IDLE;
				}
			}
			break;

		//Error state. handle errors and return to idle when errors are no longer present
		case AXIS_STATE_ERROR:

			strcpy((char*)&t->pInterface->Status.AxisState, "Machine In Error");

			t->pInterface->Commands.ToMapp.Home = 0;
			t->pInterface->Commands.Init = 0;
			t->pInterface->Commands.RequestJogNeg = 0;
			t->pInterface->Commands.RequestJogPos = 0;
			t->pInterface->Commands.RequestMoveAbs = 0;
			t->pInterface->Commands.RequestMoveAdditive = 0;
			t->pInterface->Commands.RequestHome = 0;
			t->pInterface->Commands.RequestCoupleToMaster = 0;
			t->pInterface->Commands.RequestMoveVelocity = 0;
			t->pInterface->Commands.ToMapp.JogNeg = 0;
			t->pInterface->Commands.ToMapp.JogPos = 0;
			t->pInterface->Commands.ToMapp.Home = 0;
			t->pInterface->Commands.ToMapp.MoveAbs = 0;
			t->pInterface->Commands.ToMapp.MoveVelocity = 0;
			t->pInterface->Commands.ToMapp.MoveAdditive = 0;
			t->pInterface->Commands.MoveVelocityTrigStop = 0;
			t->pInterface->Commands.ToMapp.CoupleToMaster = 0;
			t->pInterface->Commands.ToMapp.SaveConfig = 1;

			if(t->pInterface->Status.InMotion == 0){
				t->pInterface->Commands.ToMapp.Power = 0;
			}

			if(t->AlarmActive == 0)
			{
				//t->state = AXIS_STATE_INIT;
				t->state = 0; //go to whatever state 0 is for now. appropriate state should probably depend on how far we got through init process
			}

			break;
	}

	//handle drive time out because it will not become ready
	t->DriveReadyTimeout.PT = 20000;  //wait 20 seconds for drive to become ready before timing out.
	TON(&t->DriveReadyTimeout);
}
```

### Library Logical/Libraries/Lib_PBFlx (IEC)

#### FB_NDSN_MB_PBFlex_CtrlSts.st
```iecst
(* ProblueFlex Function Block for ModbusTCP *)
FUNCTION_BLOCK FB_NDSN_MB_PBFlex_CtrlSts
//******************************************************************************************************************
//Reading Section
//******************************************************************************************************************
	IF IN_b_Enable THEN
		//***************
		//Predefinition
		//***************
		i_StartAddressInput := 0;
		i_StartAddressOutput := 1024;
		i_nrRegisters := 64;
		i_datasize := 128;

		//*************************************************
		//Constant read 64 words Input buffer
		//*************************************************
		FB_AcycRead(enable := TRUE,
		pStation:= ADR(IN_mb_station),
		startAddress := i_StartAddressInput,
		nrRegisters := i_nrRegisters,
		pData := ADR(IO_Input),
		dataSize := i_datasize);
		ui_AcycRdStatus := FB_AcycRead.status;

		Melter.b_r_SystemReady := IO_Input[0].0;
		Melter.b_r_Fault := IO_Input[0].1;
		Melter.b_r_Alert := IO_Input[0].2;
		Melter.b_r_Stop := IO_Input[0].3;

		Melter.b_r_HeatersOn := IO_Input[8].0;
		Melter.b_r_StandbyOn := IO_Input[8].1;
		Melter.b_r_TemperatureAlert := IO_Input[8].2;
		Melter.b_r_TemperatureFault := IO_Input[8].3;
		Melter.b_r_TemperatureReady := IO_Input[8].4;

		Melter.b_r_TankLevelEmpty := IO_Input[12].0;
		Melter.b_r_TankLevelLow := IO_Input[12].1;
		Melter.b_r_FillSysAlert := IO_Input[12].2;
		Melter.b_r_FillSysFault := IO_Input[12].3;
		Melter.b_r_Filling := IO_Input[12].4;
		Melter.b_r_LidOpen := IO_Input[12].5;
		Melter.b_r_PumpEnabled := IO_Input[4].1;
		Melter.b_r_PumpRunning := IO_Input[4].2;
		Melter.b_r_Purging := IO_Input[4].3;
		Melter.b_r_EmptyCalibrated := IO_Input[12].6;

		tm_Command(IN := Melter.b_w_CalibrateEmpty OR Melter.b_w_ClearAlertFault , PT:= T#500MS);
		IF tm_Command.Q AND b_CommandTimerRising THEN
			Melter.b_w_ClearAlertFault :=0;
			Melter.b_w_CalibrateEmpty :=0;
		END_IF
		b_CommandTimerRising :=NOT tm_Command.Q;
		//Clear alert fault
		IO_Output[0].0 := Melter.b_w_ClearAlertFault;
		IO_Output[12].0 := Melter.b_w_ManualFill;
		IO_Output[4].3 := Melter.b_w_Purge;
		IO_Output[12].2 := Melter.b_w_CalibrateEmpty;

		//********************************************************************
		// Heater On Control Bit Logic
		//********************************************************************
		//***************************************************************************************
		// This section means if see the following edge of b_r_HeatOn, Turn off heater
		//****************************************************************************************
		tm_HeaterOff(IN := NOT Melter.b_r_HeatersOn,
		PT := t#200ms);
		b_HeaterOff := tm_HeaterOff.Q;
		IF b_HeaterOff AND b_Temp1 THEN
			b_HeaterOn := 0;
		END_IF;
		b_Temp1 := NOT b_HeaterOff;
		//***********************************************************
		// This section means if see the Rising edge of b_r_HeatOn
		// Then turn the heater on
		//***********************************************************
		IF Melter.b_r_HeatersOn AND b_Temp2 THEN
			b_HeaterOn := 1;
		END_IF;
		b_Temp2 := NOT Melter.b_r_HeatersOn;
		//***************************************************
		//Turn ON or OFF based on status of Heater
		//***************************************************
		IF NOT Melter.b_r_HeatersOn AND Melter.b_w_HeatersOnOff THEN
			b_HeaterOn := 1;
		END_IF;

		IF Melter.b_r_HeatersOn AND Melter.b_w_HeatersOnOff THEN
			b_HeaterOn := 0;
		END_IF;
		IF Melter.b_r_Fault OR Melter.b_r_TemperatureFault THEN
			b_HeaterOn := 0;
		END_IF;
		//***************************************************************
		//Below logic is to prevent HeaterOn or HeaterOff stuck situation
		//***************************************************************
		tm_HeaterOnStuck(IN := (NOT Melter.b_r_HeatersOn) AND b_HeaterOn, PT:= T#3000MS);
		b_HeaterOnStuck := tm_HeaterOnStuck.Q;

		tm_HeaterOffStuck(IN := Melter.b_r_HeatersOn AND NOT b_HeaterOn , PT:= T#3000MS);
		b_HeaterOffStuck := tm_HeaterOffStuck.Q;

		IF b_HeaterOnStuck AND b_HeaterOn THEN
			b_HeaterOn :=0;
			b_HeaterOnStuck:=0;
		END_IF;
		IF b_HeaterOffStuck AND NOT b_HeaterOn THEN
			b_HeaterOn :=1;
			b_HeaterOffStuck:=0;
		END_IF;
		//**********************************************************************
		//To generate the pulsing signal for b_w_HeatersOnOff, Turn it off here.
		//**********************************************************************
		IF Melter.b_w_HeatersOnOff THEN
			Melter.b_w_HeatersOnOff := 0;
		END_IF;
		IO_Output[8].0 := b_HeaterOn;

		//*************************************************************************************************************************
		//Pump Control Bit logic
		//*************************************************************************************************************************
		tm_PumpOff(IN := NOT Melter.b_r_PumpEnabled,
		PT := t#200ms);
		b_PumpOff := tm_PumpOff.Q;
		IF NOT Melter.b_r_PumpEnabled AND Melter.b_w_PumpOnOff AND NOT Melter.b_r_StandbyOn THEN
			b_PumpOn := 1;
		END_IF;
		IF Melter.b_r_PumpEnabled AND Melter.b_w_PumpOnOff THEN
			b_PumpOn := 0;
		END_IF;
		//******************************************************
		//Prevent turn pump on when in standby mode, othersise
		//the b_pumpon bit will stay on
		//******************************************************
		IF Melter.b_r_StandbyOn OR b_HeaterOff OR Melter.b_r_Stop THEN
			b_PumpOn := 0;
		END_IF;

		//***********************************************************************************
		//This section is to set the pump on bit on when Melter pump is turned on by itself
		//***********************************************************************************
		IF Melter.b_r_PumpEnabled AND b_Temp3 THEN
			b_PumpOn := 1;
		END_IF;
		b_Temp3 := NOT Melter.b_r_PumpEnabled;
		IF b_PumpOff AND b_Temp4 THEN
			b_PumpOn := 0;
		END_IF;
		b_Temp4 := NOT b_PumpOff;
		//***************************************************************
		//Below logic is to prevent PumpOn or PumpOff stuck situation
		//***************************************************************
		tm_PumpOnStuck(IN := (NOT Melter.b_r_PumpEnabled) AND b_PumpOn, PT:= T#3000MS);
		b_PumpOnStuck := tm_PumpOnStuck.Q;

		tm_PumpOffStuck(IN := (Melter.b_r_PumpEnabled) AND NOT b_PumpOn , PT:= T#3000MS);
		b_PumpOffStuck := tm_PumpOffStuck.Q;

		IF b_PumpOnStuck AND b_PumpOn THEN
			b_PumpOn :=0;
			b_PumpOnStuck:=0;
		END_IF;
		IF b_PumpOffStuck AND NOT b_PumpOn THEN
			b_PumpOn :=1;
			b_PumpOffStuck:=0;
		END_IF;
		//**********************************************************************
		//To generate the pulsing signal for b_w_PumpOnOff, Turn it off here.
		//**********************************************************************
		IF Melter.b_w_PumpOnOff THEN
			Melter.b_w_PumpOnOff := 0;
		END_IF;
		IO_Output[4].1 := b_PumpOn;

		//********************************************************************************************************************************
		//Standby Logic
		//********************************************************************************************************************************
		tm_StandbyOff(IN := NOT Melter.b_r_StandbyOn,
		PT := t#200ms);
		b_StandbyOff := tm_StandbyOff.Q;
		IF b_StandbyOff AND b_Temp5 THEN
			b_StandbyOn := 0;
		END_IF;
		b_Temp5 := NOT b_StandbyOff;

		IF Melter.b_r_StandbyOn AND b_Temp6 THEN
			b_StandbyOn := 1;
		END_IF;
		b_Temp6 := NOT Melter.b_r_StandbyOn;

		IF b_HeaterOff OR Melter.b_r_Fault THEN
			b_StandbyOn := 0;
		END_IF;
		//*****************************************************************************
		//This section is to determine the standby output based on the status of melter
		//with the rising edge standby on command b_w_StandbyOnOff.
		//*****************************************************************************
		IF (Melter.b_r_HeatersOn OR Melter.b_r_TemperatureReady) AND (NOT Melter.b_r_StandbyOn) AND (Melter.b_w_StandbyOnOff) THEN
			b_StandbyOn := 1;
		END_IF;

		IF (Melter.b_r_StandbyOn) AND (Melter.b_w_StandbyOnOff) THEN
			b_StandbyOn := 0;
		END_IF;
		//Below logic is to prevent StandbyOn or StandbyOff stuck situation
		tm_StandbyOnStuck(IN := (NOT Melter.b_r_StandbyOn) AND b_StandbyOn , PT:= T#3000MS);
		b_StandbyOnStuck := tm_StandbyOnStuck.Q;

		tm_StandbyOffStuck(IN := Melter.b_r_StandbyOn AND NOT b_StandbyOn, PT:= T#3000MS);
		b_StandbyOffStuck := tm_StandbyOffStuck.Q;
		IF b_StandbyOnStuck AND b_StandbyOn THEN
			b_StandbyOn :=0;
			b_StandbyOnStuck:=0;
		END_IF;
		IF b_HeaterOffStuck AND NOT b_StandbyOn THEN
			b_StandbyOn :=1;
			b_StandbyOffStuck:=0;
		END_IF;
		//**********************************************************************
		//To generate the pulsing signal for b_w_PumpOnOff, Turn it off here.
		//**********************************************************************
		IF Melter.b_w_StandbyOnOff THEN
			Melter.b_w_StandbyOnOff := 0;
		END_IF;
		IO_Output[8].1 := b_StandbyOn;

		FB_AcycWrite(enable := TRUE,
			pStation:= ADR(IN_mb_station),
			startAddress := i_StartAddressOutput,
			nrRegisters := i_nrRegisters,
			pData := ADR(IO_Output),
			dataSize := i_datasize);
			ui_AcycWtStatus := FB_AcycWrite.status;
	END_IF;
END_FUNCTION_BLOCK
```

#### FB_NDSN_MB_PBFlex_Process.st
```iecst
(* TODO: Add your comment here *)
FUNCTION_BLOCK FB_NDSN_MB_PBFlex_Process
IF IN_b_Enable THEN
	st_ADI_List[0].ui_ADI :=11682;st_ADI_List[0].ui_Size := 18;//Temperature Setpoint Aggregate(Read/Write)
	st_ADI_List[1].ui_ADI :=11683;st_ADI_List[1].ui_Size :=18;//Activate zones(Read/Write)
	st_ADI_List[2].ui_ADI :=10853;st_ADI_List[2].ui_Size := 1;//Global Standby Delta(Read/Write)
	st_ADI_List[3].ui_ADI :=10855;st_ADI_List[3].ui_Size := 1;//Manusl Standby Duration(Read/Write)
	st_ADI_List[4].ui_ADI :=10858;st_ADI_List[4].ui_Size := 1;//Auto Enter Standby Time(Read/Write)
	st_ADI_List[5].ui_ADI :=10859;st_ADI_List[5].ui_Size := 1;//Auto Heater Off Time(Read/Write)
	st_ADI_List[6].ui_ADI :=10860;st_ADI_List[6].ui_Size := 1;///Auto Standby Source(Read/Write)
	st_ADI_List[7].ui_ADI :=11376;st_ADI_List[7].ui_Size := 1;//Under Temperature Delta(Read/Write)
	st_ADI_List[8].ui_ADI :=11378;st_ADI_List[8].ui_Size := 1;//Over Temperature Delta(Read/Write)
	st_ADI_List[9].ui_ADI :=10002;st_ADI_List[9].ui_Size := 1;//Temperature Unit	(Read/Write)
	st_ADI_List[10].ui_ADI :=10547;st_ADI_List[10].ui_Size := 1;//Global Temperature Setpoint(Read/Write)
	st_ADI_List[11].ui_ADI :=10549;st_ADI_List[11].ui_Size := 1;//Global Hose Setpoint(Read/Write)
	st_ADI_List[12].ui_ADI :=10548;st_ADI_List[12].ui_Size := 1;//Global Gun Setpoint(Read/Write)
	st_ADI_List[13].ui_ADI :=6102;st_ADI_List[13].ui_Size := 1;//Pressure Unit(Read/Write)
	st_ADI_List[14].ui_ADI :=6203;st_ADI_List[14].ui_Size := 2;//Pressure Setpoint(Read/Write)
	st_ADI_List[15].ui_ADI :=6946;st_ADI_List[15].ui_Size := 2;//Max Pressure limit(Read/Write)
	st_ADI_List[16].ui_ADI :=7046;st_ADI_List[16].ui_Size := 2;//Min Pressure Limit(Read/Write)
	st_ADI_List[17].ui_ADI :=7148;st_ADI_List[17].ui_Size := 2;//Under Pressure Delta(Read/Write)
	st_ADI_List[18].ui_ADI :=7248;st_ADI_List[18].ui_Size := 2;//Over Pressure Delta(Read/Write)
	st_ADI_List[19].ui_ADI :=7146;st_ADI_List[19].ui_Size := 1;//Enable Pressure High low Limit(Read/Write)
	st_ADI_List[20].ui_ADI :=7147;st_ADI_List[20].ui_Size := 1;//Enable Hydraulic Scaling(Read/Write)
	st_ADI_List[21].ui_ADI :=13017;st_ADI_List[21].ui_Size := 1;//Enable Fill(Read/Write)
	st_ADI_List[22].ui_ADI :=13003;st_ADI_List[22].ui_Size := 1;//Target Fill Level(Read/Write)
	st_ADI_List[23].ui_ADI :=13008;st_ADI_List[23].ui_Size := 1;//Max Fill Time(Read/Write)
	st_ADI_List[24].ui_ADI :=13009;st_ADI_List[24].ui_Size := 1;//Alert Stop Delay Time(Read/Write)
	st_ADI_List[25].ui_ADI :=13010;st_ADI_List[25].ui_Size := 1;//Low Level Threshold(Read/Write)
	st_ADI_List[26].ui_ADI :=13012;st_ADI_List[26].ui_Size := 1;//Lid Open Alert Time(Read/Write)
	st_ADI_List[27].ui_ADI :=13018;st_ADI_List[27].ui_Size := 1;//Alert Stop Delay Time(Read/Write)
	st_ADI_List[28].ui_ADI :=801;st_ADI_List[28].ui_Size := 1;//Enable Auto Pump(Read/Write)
	st_ADI_List[29].ui_ADI :=19;st_ADI_List[29].ui_Size := 1;//Temperature Ready Delay Time(Read/Write)
	st_ADI_List[30].ui_ADI :=22;st_ADI_List[30].ui_Size := 1;//Mass Unit(Read/Write)
	st_ADI_List[31].ui_ADI :=11681;st_ADI_List[31].ui_Size := 18;//Actual Temperature(Read Only)
	st_ADI_List[32].ui_ADI :=11685;st_ADI_List[32].ui_Size := 18;//Temperature Status(Read Only)
	st_ADI_List[33].ui_ADI :=6103;st_ADI_List[33].ui_Size := 2;//Actual Pressure Value(Read Only)
	st_ADI_List[34].ui_ADI :=6002;st_ADI_List[34].ui_Size := 1;//Pressure Sensor Alarm(Read Only)
	st_ADI_List[35].ui_ADI :=13002;st_ADI_List[35].ui_Size := 1;//Actual Fill Level(Read Only)
	st_ADI_List[36].ui_ADI :=29;st_ADI_List[36].ui_Size := 1;//Current Fault Code(Read Only)
	st_ADI_List[37].ui_ADI :=13;st_ADI_List[37].ui_Size := 1;//Software Version(Read Only)
	st_ADI_List[38].ui_ADI :=16;st_ADI_List[38].ui_Size := 2;//Operation Hours(Read Only)
	st_ADI_List[39].ui_ADI :=30;st_ADI_List[39].ui_Size := 4;//Inventory	(Read Only)

	//System Inventory
	Melter.st_r_Devices.b_r_TempCtrl_Board1 := Melter.i_r_Gen_arr_SysInventory[0].0;
	Melter.st_r_Devices.b_r_TempCtrl_Board2 := Melter.i_r_Gen_arr_SysInventory[0].1;
	Melter.st_r_Devices.b_r_TempCtrl_Board3 := Melter.i_r_Gen_arr_SysInventory[0].2;
	Melter.st_r_Devices.b_r_TempCtrl_Board4 := Melter.i_r_Gen_arr_SysInventory[0].3;
	Melter.st_r_Devices.b_r_OEM_Unit:= Melter.i_r_Gen_arr_SysInventory[0].8;
	Melter.st_r_Devices.b_r_OLED_Unit:= Melter.i_r_Gen_arr_SysInventory[0].9;
	Melter.st_r_Devices.b_r_WIFI_Board:= Melter.i_r_Gen_arr_SysInventory[0].10;
	Melter.st_r_Devices.b_r_Refill_Board:= Melter.i_r_Gen_arr_SysInventory[0].11;
	Melter.st_r_Devices.b_r_Anybus_Board:= Melter.i_r_Gen_arr_SysInventory[0].12;
	Melter.st_r_Devices.b_r_Press_Sensor:= Melter.i_r_Gen_arr_SysInventory[0].14;
	Melter.st_r_Devices.b_r_Press_CtrlValve:= Melter.i_r_Gen_arr_SysInventory[0].15;
	Melter.st_r_Devices.i_r_NumOfTempZones_External:= Melter.i_r_Gen_arr_SysInventory[1]/256;
	Melter.st_r_Devices.i_r_NumOfTempZones_Internal:= Melter.i_r_Gen_arr_SysInventory[1]-Melter.st_r_Devices.i_r_NumOfTempZones_External*256;
	Melter.st_r_Devices.i_r_NumOfPumps:= Melter.i_r_Gen_arr_SysInventory[2]/256;
	Melter.st_r_Devices.i_r_NumOfMotors:= Melter.i_r_Gen_arr_SysInventory[2]-Melter.st_r_Devices.i_r_NumOfPumps*256;
	Melter.st_r_Devices.i_r_NumOfWebClients := Melter.i_r_Gen_arr_SysInventory[3]/256;
	Melter.st_r_Devices.i_r_NumOfATS:= Melter.i_r_Gen_arr_SysInventory[3]-Melter.st_r_Devices.i_r_NumOfWebClients*256;

	i_ADI_Range := 0;
	FOR i := 0 TO i_rwADI_Count  DO
		i_ADI_Range:= i_ADI_Range + UDINT_TO_INT(st_ADI_List[i].ui_Size);
		arr_WriteIndex[i] := i_ADI_Range;//Index of all Read/Write ADI
		arr_WriteStartingAddress[i + 1] := i_ADI_Range;//All Read/Write ADI Starting Address
	END_FOR;

		//*************************************************
		//Create Reading Tick to Acyclic Read, Acyc Read
		//Start when timer is triggered ends when all
		//Acyc data are red, then wait for next Timer cycle
		//*************************************************
	tm_Acyc(IN := NOT b_read,
	PT := T#2000MS);
	b_read := tm_Acyc.Q ;

	//******************************************************************
	//Sequentially read ALL ADIs and store into structure
	//b_read will initiate when tm_Acyc Expired,b_AcycRD_Tick will
	//trigger the funciton block when read is done,
	//b_AcycRD_Enable only last during Acyclic reading in process
	//When last ADI been read, it will stop reading until next cycle
	//*******************************************************************
	FB_AcycRead_Para(enable := TRUE,
		pStation:= ADR(IN_mb_station),
		startAddress := st_ADI_List[i_Index].ui_ADI,
		nrRegisters := st_ADI_List[i_Index].ui_Size,
		pData := ADR(arr_ResponseValue),
		dataSize := st_ADI_List[i_Index].ui_Size*2);
	ui_AcycRdStatus_Para := FB_AcycRead_Para.status;
	b_AcycRD_Tick := FALSE;
	b_AcycRD_Done := FALSE;
	//*******************************************************************
	//Below is the section handling pressure reading, since the pressure
	//over fieldbus is always in PSI, the following logic will convert
	//Pressure value into different value based on the value setting
	//*******************************************************************
	i_ADI := st_ADI_List[i_Index].ui_ADI;
	i_Size := UDINT_TO_INT(st_ADI_List[i_Index].ui_Size);
	IF ui_AcycRdStatus_Para <>65535 AND b_AcycRdDnRising THEN
		b_AcycRD_Done := TRUE;
	END_IF;
	b_AcycRdDnRising := (ui_AcycRdStatus_Para = 65535);
	IF b_AcycRD_Done THEN
		brsmemcpy(pDest:=ADR(arr_HMI[i_ValueIndex]) , pSrc:= ADR(arr_ResponseValue) , length:=i_Size*2 );
		IF i_Size = 2 THEN
			arr_i_DW_Temp[0] := arr_ResponseValue[0];
			arr_i_DW_Temp[1] := arr_ResponseValue[1];
			//Convert the unit based on pressure unit read from melter
			IF (i_ADI > 6000) AND (i_ADI < 8000) THEN
				brsmemcpy(pDest:=ADR(di_Press) , pSrc:= ADR(arr_ResponseValue) , length:=4 );
				//di_Press := arr_ResponseValue[0]+65536*arr_ResponseValue[1];
				CASE Melter.i_rw_Press_Unit OF
					0://psi
						r_Press := UDINT_TO_REAL(di_Press) / 1000.000;
					1://kpa
						r_Press := UDINT_TO_REAL(di_Press) / 145.0377377;
					2://bar
						r_Press := UDINT_TO_REAL(di_Press) / 14503.77377;
				END_CASE;
				brsmemcpy(pDest:=ADR(arr_i_DW_Temp[0]) , pSrc:= ADR(r_Press) , length:=4 );
				arr_HMI[i_ValueIndex] := arr_i_DW_Temp[0];
				arr_HMI[i_ValueIndex+1 ] := arr_i_DW_Temp[1];
			ELSE
				arr_HMI[i_ValueIndex] := arr_i_DW_Temp[0];
				arr_HMI[i_ValueIndex+1 ] := arr_i_DW_Temp[1];
			END_IF
		END_IF;
		//****************************************************
		//After reading the current ADI, index to next one
		//****************************************************
		i_ValueIndex := i_ValueIndex + UDINT_TO_INT(st_ADI_List[i_Index].ui_Size);
		i_Index := i_Index + 1;
	END_IF;

	//****************************************************
	//Copy all reading value into structure
	//****************************************************
	IF b_read THEN
		brsmemcpy(pDest:=ADR(Melter.i_rw_Temp_arr_ZoneSP[0]) , pSrc:= ADR(arr_HMI[0]) , length:=i_SizeofStruct);
		brsmemcpy(pDest:=ADR(arr_HMI_Buffer[0]) , pSrc:= ADR(arr_HMI[0]) , length:=i_rwDataSize*2 );
	END_IF;

	//*******************************************************
	//When finish the last ADI, Rest until next reding cycle
	//*******************************************************
	IF i_Index = i_ADI_Size  THEN
		i_Index := 0;
		b_AcycRD_Enable :=FALSE;
		i_ValueIndex :=0;
		b_AcycWT_Start :=0;
	END_IF;
	//**********************************************************************************************
	//Copy all read/write ADI reading into arr_HMI_Buffer_Compare for further generating Write Event
	//***********************************************************************************************
	brsmemcpy(pDest:=ADR(arr_HMI_Compare[0]) , pSrc:= ADR(Melter.i_rw_Temp_arr_ZoneSP[0]) ,length:=i_rwDataSize*2 );
END_IF;

	//**************************************************************************************
	//Compare arr_HMI_Compare with arr_HMI_Buffer to generate write event
	//**************************************************************************************
	tm_WriteEvent(IN :=b_WriteEvent,
		PT := T#300MS);
	IF tm_WriteEvent.Q OR (b_AcycWT_Done AND b_AcycWT_Rising) THEN
		b_WriteEvent :=0;
	END_IF;
	b_AcycWT_Rising := NOT b_AcycWT_Done;

	b_WriteEventONS := 0;
	FOR i:=0 TO i_rwDataSize-1 BY 1 DO
		IF (arr_HMI_Compare[i] <> arr_HMI_Buffer[i]) AND NOT b_AcycWT_Start THEN
			i_CompareIndex := i;
			b_WriteEvent := TRUE;
			b_WriteEventONS := TRUE;
			arr_HMI_Buffer[i] :=arr_HMI_Compare[i];
			b_AcycWT_Start :=1;
			i_wttest := i_wttest +1;
			EXIT;
		END_IF;
	END_FOR;

	IF (b_AcycWT_Done OR tm_WriteEvent.Q)AND b_AcycWT_DN_Rising THEN
		b_AcycWT_Start :=0;
	END_IF;
	b_AcycWT_DN_Rising:= NOT (b_AcycWT_Done OR tm_WriteEvent.Q);

	IF b_WriteEventONS THEN
		//***************************************************************
		//When write event locate the write index inside arr_WriteIndex
		//***************************************************************
		FOR i := 0 TO i_rwADI_Count DO
			IF i_CompareIndex < arr_WriteIndex[i] THEN
				i_Index_Write := i;
				EXIT;
			END_IF;
		END_FOR;
		//***************************************************************
		//If pressure ADI generate write event, conver the unit back to PSI
		//***************************************************************
		i_writesize := UDINT_TO_INT(st_ADI_List[i_Index_Write].ui_Size);
		IF i_writesize = 2 THEN
			brsmemcpy(pDest:=ADR(r_PressConvert) , pSrc:= ADR(arr_HMI_Compare[arr_WriteStartingAddress[i_Index_Write]]) , length:=4 );
			CASE Melter.i_rw_Press_Unit OF
				0://psi
					di_Press_psi := REAL_TO_UDINT(r_PressConvert * 1000.000);
				1://kpa
					di_Press_psi :=REAL_TO_UDINT( r_PressConvert* 145.0377377);
				2://bar
					di_Press_psi := REAL_TO_UDINT(r_PressConvert* 14503.77377);
			END_CASE;
			brsmemcpy(pDest:=ADR(arr_di_Press_psi[0]) , pSrc:= ADR(di_Press_psi) , length:=4 );
			i_arr_WriteBuffer[0] := arr_di_Press_psi[0];
			i_arr_WriteBuffer[1] := arr_di_Press_psi[1];
			brsmemcpy(pDest:=ADR(arr_HMI[arr_WriteStartingAddress[i_Index_Write]]) , pSrc:= ADR(arr_HMI_Compare[arr_WriteStartingAddress[i_Index_Write]]) , length:=4);
		ELSE
			brsmemcpy(pDest:=ADR(i_arr_WriteBuffer[0]) , pSrc:= ADR(arr_HMI_Compare[arr_WriteStartingAddress[i_Index_Write]]) , length:=i_writesize*2);
			brsmemcpy(pDest:=ADR(arr_HMI[arr_WriteStartingAddress[i_Index_Write]]) , pSrc:= ADR(arr_HMI_Compare[arr_WriteStartingAddress[i_Index_Write]]) , length:=i_writesize*2);
		END_IF;
	END_IF;
	//Acyclic Write Function block
	FB_AcycWrite(enable := b_WriteEvent,
		pStation:= ADR(IN_mb_station),
		startAddress := st_ADI_List[i_Index_Write].ui_ADI,
		nrRegisters := st_ADI_List[i_Index_Write].ui_Size,
		pData := ADR(i_arr_WriteBuffer),
		dataSize := st_ADI_List[i_Index_Write].ui_Size*2);
	ui_AcycWtStatus := FB_AcycWrite.status;

	b_AcycWT_Done := FALSE;
	IF ui_AcycWtStatus <>65535 AND b_AcycWTDnRising THEN
		b_AcycWT_Done := TRUE;
	END_IF;
	b_AcycWTDnRising := (ui_AcycWtStatus = 65535);

END_FUNCTION_BLOCK
```
